LIN {X 0,Y 501.495,Z 927.191,A -85,B 0,C 180,E1 14910.89,E2 14910.89} C_VEL
LIN {X 0,Y 476.741,Z 888.568,A -85,B 0,C 180,E1 14918.992,E2 14918.992} C_VEL
LIN {X 0,Y 459.302,Z 865.995,A -85,B 0,C 180,E1 14927.264,E2 14927.264} C_VEL
LIN {X 0,Y 453.825,Z 859.085,A -85,B 0,C 180,E1 14931.559,E2 14931.559} C_VEL
LIN {X 0,Y 449.713,Z 853.483,A -85,B 0,C 180,E1 14939.969,E2 14939.969} C_VEL
LIN {X 0,Y 456.227,Z 862.461,A -85,B 0,C 180,E1 14950.385,E2 14950.385} C_VEL
LIN {X 0,Y 467.484,Z 876.849,A -85,B 0,C 180,E1 14956.99,E2 14956.99} C_VEL
LIN {X 0,Y 488.733,Z 906.336,A -85,B 0,C 180,E1 14964.926,E2 14964.926} C_VEL
LIN {X 0,Y 513.325,Z 949.109,A -85,B 0,C 180,E1 14972.183,E2 14972.183} C_VEL
LIN {X 0,Y 525.687,Z 980.917,A -85,B 0,C 180,E1 14976.061,E2 14976.061} C_VEL
LIN {X 0,Y 510.224,Z 1051.4,A -85,B 0,C 180,E1 14979.425,E2 14979.425} C_VEL
LIN {X 0,Y 490.436,Z 1119.326,A -85,B 0,C 180,E1 14984.666,E2 14984.666} C_VEL
LIN {X 0,Y 470.634,Z 1178.94,A -85,B 0,C 180,E1 14991.825,E2 14991.825} C_VEL
LIN {X 0,Y 455.077,Z 1227.051,A -85,B 0,C 180,E1 15000.689,E2 15000.689} C_VEL
LIN {X 0,Y 446.421,Z 1260.098,A -85,B 0,C 180,E1 15010.141,E2 15010.141} C_VEL
LIN {X 0,Y 443.545,Z 1278.907,A -85,B 0,C 180,E1 15019.161,E2 15019.161} C_VEL
LIN {X 0,Y 443.233,Z 1286.226,A -85,B 0,C 180,E1 15027.058,E2 15027.058} C_VEL
LIN {X 0,Y 443.148,Z 1285.182,A -85,B 0,C 180,E1 15034.908,E2 15034.908} C_VEL
LIN {X 0,Y 443.658,Z 1277.124,A -85,B 0,C 180,E1 15041.963,E2 15041.963} C_VEL
LIN {X 0,Y 437.23,Z 1269.245,A -85,B 0,C 180,E1 15046.394,E2 15046.394} C_VEL
LIN {X 0,Y 443.661,Z 1240.734,A -85,B 0,C 180,E1 15056.383,E2 15056.383} C_VEL
LIN {X 0,Y 457.28,Z 1198.235,A -85,B 0,C 180,E1 15065.684,E2 15065.684} C_VEL
LIN {X 0,Y 476.969,Z 1142.146,A -85,B 0,C 180,E1 15073.629,E2 15073.629} C_VEL
LIN {X 0,Y 497.802,Z 1076.976,A -85,B 0,C 180,E1 15079.607,E2 15079.607} C_VEL
LIN {X 0,Y 516.277,Z 1003.643,A -85,B 0,C 180,E1 15083.798,E2 15083.798} C_VEL
LIN {X 0,Y 519.992,Z 980.36,A -85,B 0,C 180,E1 15084.85,E2 15084.85} C_VEL
LIN {X 0,Y 499.484,Z 935.129,A -85,B 0,C 180,E1 15091.226,E2 15091.226} C_VEL
LIN {X 0,Y 476.703,Z 899.572,A -85,B 0,C 180,E1 15098.748,E2 15098.748} C_VEL
LIN {X 0,Y 458.796,Z 874.684,A -85,B 0,C 180,E1 15107.256,E2 15107.256} C_VEL
LIN {X 0,Y 451.996,Z 866.689,A -85,B 0,C 180,E1 15112.801,E2 15112.801} C_VEL
LIN {X 0,Y 448.923,Z 862.376,A -85,B 0,C 180,E1 15120.515,E2 15120.515} C_VEL
LIN {X 0,Y 454.937,Z 870.236,A -85,B 0,C 180,E1 15130.114,E2 15130.114} C_VEL
LIN {X 0,Y 466.224,Z 885.028,A -85,B 0,C 180,E1 15136.938,E2 15136.938} C_VEL
LIN {X 0,Y 487.537,Z 915.75,A -85,B 0,C 180,E1 15145.24,E2 15145.24} C_VEL
LIN {X 0,Y 511.002,Z 960.348,A -85,B 0,C 180,E1 15152.735,E2 15152.735} C_VEL
LIN {X 0,Y 519.263,Z 983.911,A -85,B 0,C 180,E1 15155.652,E2 15155.652} C_VEL
LIN {X 0,Y 501.618,Z 1058.051,A -85,B 0,C 180,E1 15159.562,E2 15159.562} C_VEL
LIN {X 0,Y 480.854,Z 1124.559,A -85,B 0,C 180,E1 15165.264,E2 15165.264} C_VEL
LIN {X 0,Y 460.838,Z 1181.172,A -85,B 0,C 180,E1 15172.79,E2 15172.79} C_VEL
LIN {X 0,Y 445.644,Z 1226.459,A -85,B 0,C 180,E1 15182.124,E2 15182.124} C_VEL
LIN {X 0,Y 437.765,Z 1257.62,A -85,B 0,C 180,E1 15192.467,E2 15192.467} C_VEL
LIN {X 0,Y 435.276,Z 1273.211,A -85,B 0,C 180,E1 15201.989,E2 15201.989} C_VEL
LIN {X 0,Y 435.375,Z 1277.067,A -85,B 0,C 180,E1 15210.998,E2 15210.998} C_VEL
LIN {X 0,Y 435.467,Z 1270.726,A -85,B 0,C 180,E1 15220.028,E2 15220.028} C_VEL
LIN {X 0,Y 438.618,Z 1252.212,A -85,B 0,C 180,E1 15229.701,E2 15229.701} C_VEL
LIN {X 0,Y 448.511,Z 1217.589,A -85,B 0,C 180,E1 15239.961,E2 15239.961} C_VEL
LIN {X 0,Y 464.976,Z 1169.906,A -85,B 0,C 180,E1 15248.872,E2 15248.872} C_VEL
LIN {X 0,Y 485.246,Z 1111.113,A -85,B 0,C 180,E1 15256.017,E2 15256.017} C_VEL
LIN {X 0,Y 505.549,Z 1043.955,A -85,B 0,C 180,E1 15261.223,E2 15261.223} C_VEL
LIN {X 0,Y 518.976,Z 979.558,A -85,B 0,C 180,E1 15264.58,E2 15264.58} C_VEL
LIN {X 0,Y 496.602,Z 930.952,A -85,B 0,C 180,E1 15271.706,E2 15271.706} C_VEL
LIN {X 0,Y 473.84,Z 895.17,A -85,B 0,C 180,E1 15279.593,E2 15279.593} C_VEL
LIN {X 0,Y 457.868,Z 873.617,A -85,B 0,C 180,E1 15287.532,E2 15287.532} C_VEL
LIN {X 0,Y 452.354,Z 866.791,A -85,B 0,C 180,E1 15292.017,E2 15292.017} C_VEL
LIN {X 0,Y 448.735,Z 861.449,A -85,B 0,C 180,E1 15299.969,E2 15299.969} C_VEL
LIN {X 0,Y 455.016,Z 870.359,A -85,B 0,C 180,E1 15310.231,E2 15310.231} C_VEL
LIN {X 0,Y 466.161,Z 884.963,A -85,B 0,C 180,E1 15316.877,E2 15316.877} C_VEL
LIN {X 0,Y 487.839,Z 915.843,A -85,B 0,C 180,E1 15325.159,E2 15325.159} C_VEL
LIN {X 0,Y 511.528,Z 960.138,A -85,B 0,C 180,E1 15332.514,E2 15332.514} C_VEL
LIN {X 0,Y 520.206,Z 984.714,A -85,B 0,C 180,E1 15335.473,E2 15335.473} C_VEL
LIN {X 0,Y 503.561,Z 1056.776,A -85,B 0,C 180,E1 15339.044,E2 15339.044} C_VEL
LIN {X 0,Y 483.304,Z 1123.218,A -85,B 0,C 180,E1 15344.36,E2 15344.36} C_VEL
LIN {X 0,Y 462.993,Z 1181.823,A -85,B 0,C 180,E1 15351.633,E2 15351.633} C_VEL
LIN {X 0,Y 447.269,Z 1228.623,A -85,B 0,C 180,E1 15360.551,E2 15360.551} C_VEL
LIN {X 0,Y 438.37,Z 1261.359,A -85,B 0,C 180,E1 15370.287,E2 15370.287} C_VEL
LIN {X 0,Y 435.523,Z 1280.164,A -85,B 0,C 180,E1 15379.973,E2 15379.973} C_VEL
LIN {X 0,Y 434.878,Z 1286.595,A -85,B 0,C 180,E1 15389.001,E2 15389.001} C_VEL
LIN {X 0,Y 435.311,Z 1282.6,A -85,B 0,C 180,E1 15398.01,E2 15398.01} C_VEL
LIN {X 0,Y 437.23,Z 1269.245,A -85,B 0,C 180,E1 15406.394,E2 15406.394} C_VEL
LIN {X 0,Y 431.04,Z 1259.359,A -85,B 0,C 180,E1 15410.823,E2 15410.823} C_VEL
LIN {X 0,Y 441.547,Z 1223.978,A -85,B 0,C 180,E1 15421.056,E2 15421.056} C_VEL
LIN {X 0,Y 458.603,Z 1176.1,A -85,B 0,C 180,E1 15429.877,E2 15429.877} C_VEL
LIN {X 0,Y 479.802,Z 1116.617,A -85,B 0,C 180,E1 15437.002,E2 15437.002} C_VEL
LIN {X 0,Y 500.574,Z 1049.302,A -85,B 0,C 180,E1 15442.146,E2 15442.146} C_VEL
LIN {X 0,Y 514.628,Z 984.001,A -85,B 0,C 180,E1 15445.46,E2 15445.46} C_VEL
LIN {X 0,Y 494.654,Z 938.886,A -85,B 0,C 180,E1 15452.034,E2 15452.034} C_VEL
LIN {X 0,Y 472.061,Z 902.933,A -85,B 0,C 180,E1 15460.067,E2 15460.067} C_VEL
LIN {X 0,Y 456.456,Z 881.69,A -85,B 0,C 180,E1 15468.088,E2 15468.088} C_VEL
LIN {X 0,Y 450.6,Z 874.34,A -85,B 0,C 180,E1 15473.264,E2 15473.264} C_VEL
LIN {X 0,Y 447.949,Z 870.312,A -85,B 0,C 180,E1 15480.517,E2 15480.517} C_VEL
LIN {X 0,Y 453.804,Z 878.246,A -85,B 0,C 180,E1 15490.018,E2 15490.018} C_VEL
LIN {X 0,Y 464.959,Z 893.354,A -85,B 0,C 180,E1 15496.925,E2 15496.925} C_VEL
LIN {X 0,Y 485.315,Z 923.772,A -85,B 0,C 180,E1 15505.11,E2 15505.11} C_VEL
LIN {X 0,Y 506.806,Z 966.395,A -85,B 0,C 180,E1 15512.381,E2 15512.381} C_VEL
LIN {X 0,Y 513.595,Z 988.518,A -85,B 0,C 180,E1 15515.105,E2 15515.105} C_VEL
LIN {X 0,Y 495.036,Z 1062.693,A -85,B 0,C 180,E1 15519.15,E2 15519.15} C_VEL
LIN {X 0,Y 473.79,Z 1127.945,A -85,B 0,C 180,E1 15524.925,E2 15524.925} C_VEL
LIN {X 0,Y 453.117,Z 1184.181,A -85,B 0,C 180,E1 15532.654,E2 15532.654} C_VEL
LIN {X 0,Y 437.576,Z 1228.757,A -85,B 0,C 180,E1 15542.205,E2 15542.205} C_VEL
LIN {X 0,Y 429.704,Z 1258.601,A -85,B 0,C 180,E1 15552.543,E2 15552.543} C_VEL
LIN {X 0,Y 427.308,Z 1273.298,A -85,B 0,C 180,E1 15561.839,E2 15561.839} C_VEL
LIN {X 0,Y 427.391,Z 1277.155,A -85,B 0,C 180,E1 15571.017,E2 15571.017} C_VEL
LIN {X 0,Y 427.483,Z 1270.816,A -85,B 0,C 180,E1 15580.217,E2 15580.217} C_VEL
LIN {X 0,Y 431.216,Z 1251.295,A -85,B 0,C 180,E1 15590.462,E2 15590.462} C_VEL
LIN {X 0,Y 441.691,Z 1216.518,A -85,B 0,C 180,E1 15600.781,E2 15600.781} C_VEL
LIN {X 0,Y 458.714,Z 1169.437,A -85,B 0,C 180,E1 15609.614,E2 15609.614} C_VEL
LIN {X 0,Y 479.414,Z 1111.581,A -85,B 0,C 180,E1 15616.691,E2 15616.691} C_VEL
LIN {X 0,Y 500.553,Z 1043.74,A -85,B 0,C 180,E1 15621.972,E2 15621.972} C_VEL
LIN {X 0,Y 513.747,Z 983.715,A -85,B 0,C 180,E1 15625.133,E2 15625.133} C_VEL
LIN {X 0,Y 492.652,Z 936.614,A -85,B 0,C 180,E1 15632.236,E2 15632.236} C_VEL
LIN {X 0,Y 471.152,Z 901.763,A -85,B 0,C 180,E1 15640.147,E2 15640.147} C_VEL
LIN {X 0,Y 456.144,Z 880.962,A -85,B 0,C 180,E1 15647.999,E2 15647.999} C_VEL
LIN {X 0,Y 450.912,Z 874.489,A -85,B 0,C 180,E1 15652.478,E2 15652.478} C_VEL
LIN {X 0,Y 447.759,Z 869.4,A -85,B 0,C 180,E1 15659.969,E2 15659.969} C_VEL
LIN {X 0,Y 453.811,Z 878.238,A -85,B 0,C 180,E1 15670.076,E2 15670.076} C_VEL
LIN {X 0,Y 465.304,Z 893.818,A -85,B 0,C 180,E1 15677.032,E2 15677.032} C_VEL
LIN {X 0,Y 485.785,Z 924.152,A -85,B 0,C 180,E1 15685.088,E2 15685.088} C_VEL
LIN {X 0,Y 508.014,Z 967.632,A -85,B 0,C 180,E1 15692.348,E2 15692.348} C_VEL
LIN {X 0,Y 515.001,Z 987.452,A -85,B 0,C 180,E1 15694.839,E2 15694.839} C_VEL
LIN {X 0,Y 498.134,Z 1057.756,A -85,B 0,C 180,E1 15698.378,E2 15698.378} C_VEL
LIN {X 0,Y 477.644,Z 1122.698,A -85,B 0,C 180,E1 15703.601,E2 15703.601} C_VEL
LIN {X 0,Y 456.424,Z 1181.853,A -85,B 0,C 180,E1 15711.001,E2 15711.001} C_VEL
LIN {X 0,Y 439.967,Z 1228.53,A -85,B 0,C 180,E1 15720.013,E2 15720.013} C_VEL
LIN {X 0,Y 430.816,Z 1260.254,A -85,B 0,C 180,E1 15729.524,E2 15729.524} C_VEL
LIN {X 0,Y 427.57,Z 1278.729,A -85,B 0,C 180,E1 15738.751,E2 15738.751} C_VEL
LIN {X 0,Y 427.242,Z 1286.051,A -85,B 0,C 180,E1 15746.948,E2 15746.948} C_VEL
LIN {X 0,Y 427.152,Z 1285.007,A -85,B 0,C 180,E1 15755.092,E2 15755.092} C_VEL
LIN {X 0,Y 428.304,Z 1273.725,A -85,B 0,C 180,E1 15764.351,E2 15764.351} C_VEL
LIN {X 0,Y 431.04,Z 1259.359,A -85,B 0,C 180,E1 15770.823,E2 15770.823} C_VEL
LIN {X 0,Y 426.882,Z 1247.494,A -85,B 0,C 180,E1 15775.272,E2 15775.272} C_VEL
LIN {X 0,Y 440.642,Z 1206.475,A -85,B 0,C 180,E1 15785.339,E2 15785.339} C_VEL
LIN {X 0,Y 460.695,Z 1153.533,A -85,B 0,C 180,E1 15793.646,E2 15793.646} C_VEL
LIN {X 0,Y 483.118,Z 1089.437,A -85,B 0,C 180,E1 15800.131,E2 15800.131} C_VEL
LIN {X 0,Y 503.794,Z 1017.149,A -85,B 0,C 180,E1 15804.635,E2 15804.635} C_VEL
LIN {X 0,Y 509.483,Z 987.866,A -85,B 0,C 180,E1 15806.041,E2 15806.041} C_VEL
LIN {X 0,Y 490.493,Z 944.188,A -85,B 0,C 180,E1 15812.634,E2 15812.634} C_VEL
LIN {X 0,Y 469.524,Z 909.664,A -85,B 0,C 180,E1 15820.569,E2 15820.569} C_VEL
LIN {X 0,Y 454.853,Z 889.166,A -85,B 0,C 180,E1 15828.488,E2 15828.488} C_VEL
LIN {X 0,Y 449.46,Z 882.146,A -85,B 0,C 180,E1 15833.454,E2 15833.454} C_VEL
LIN {X 0,Y 447.012,Z 878.319,A -85,B 0,C 180,E1 15841.004,E2 15841.004} C_VEL
LIN {X 0,Y 452.674,Z 886.24,A -85,B 0,C 180,E1 15849.921,E2 15849.921} C_VEL
LIN {X 0,Y 463.901,Z 901.925,A -85,B 0,C 180,E1 15857.026,E2 15857.026} C_VEL
LIN {X 0,Y 483.881,Z 933.368,A -85,B 0,C 180,E1 15865.366,E2 15865.366} C_VEL
LIN {X 0,Y 503.989,Z 976.276,A -85,B 0,C 180,E1 15872.584,E2 15872.584} C_VEL
LIN {X 0,Y 508.188,Z 992.307,A -85,B 0,C 180,E1 15874.517,E2 15874.517} C_VEL
LIN {X 0,Y 488.734,Z 1066.589,A -85,B 0,C 180,E1 15878.677,E2 15878.677} C_VEL
LIN {X 0,Y 466.613,Z 1131.769,A -85,B 0,C 180,E1 15884.628,E2 15884.628} C_VEL
LIN {X 0,Y 445.395,Z 1187.175,A -85,B 0,C 180,E1 15892.51,E2 15892.51} C_VEL
LIN {X 0,Y 429.653,Z 1230.659,A -85,B 0,C 180,E1 15902.183,E2 15902.183} C_VEL
LIN {X 0,Y 421.726,Z 1259.366,A -85,B 0,C 180,E1 15912.523,E2 15912.523} C_VEL
LIN {X 0,Y 419.26,Z 1274.237,A -85,B 0,C 180,E1 15922.727,E2 15922.727} C_VEL
LIN {X 0,Y 419.385,Z 1277.242,A -85,B 0,C 180,E1 15931.036,E2 15931.036} C_VEL
LIN {X 0,Y 419.52,Z 1270.906,A -85,B 0,C 180,E1 15940.413,E2 15940.413} C_VEL
LIN {X 0,Y 423.479,Z 1251.584,A -85,B 0,C 180,E1 15950.771,E2 15950.771} C_VEL
LIN {X 0,Y 434.477,Z 1216.776,A -85,B 0,C 180,E1 15961.305,E2 15961.305} C_VEL
LIN {X 0,Y 452.135,Z 1169.99,A -85,B 0,C 180,E1 15970.217,E2 15970.217} C_VEL
LIN {X 0,Y 473.478,Z 1112.488,A -85,B 0,C 180,E1 15977.338,E2 15977.338} C_VEL
LIN {X 0,Y 495.08,Z 1045.523,A -85,B 0,C 180,E1 15982.61,E2 15982.61} C_VEL
LIN {X 0,Y 508.615,Z 988.345,A -85,B 0,C 180,E1 15985.617,E2 15985.617} C_VEL
LIN {X 0,Y 488.905,Z 942.436,A -85,B 0,C 180,E1 15992.727,E2 15992.727} C_VEL
LIN {X 0,Y 468.545,Z 908.479,A -85,B 0,C 180,E1 16000.647,E2 16000.647} C_VEL
LIN {X 0,Y 454.199,Z 887.857,A -85,B 0,C 180,E1 16008.652,E2 16008.652} C_VEL
LIN {X 0,Y 449.303,Z 881.947,A -85,B 0,C 180,E1 16013.182,E2 16013.182} C_VEL
LIN {X 0,Y 446.773,Z 877.479,A -85,B 0,C 180,E1 16020.212,E2 16020.212} C_VEL
LIN {X 0,Y 452.748,Z 886.334,A -85,B 0,C 180,E1 16030.039,E2 16030.039} C_VEL
LIN {X 0,Y 466.383,Z 904.689,A -85,B 0,C 180,E1 16038.09,E2 16038.09} C_VEL
LIN {X 0,Y 488.354,Z 940.813,A -85,B 0,C 180,E1 16046.7,E2 16046.7} C_VEL
LIN {X 0,Y 508.381,Z 985.693,A -85,B 0,C 180,E1 16053.642,E2 16053.642} C_VEL
LIN {X 0,Y 508.76,Z 994.841,A -85,B 0,C 180,E1 16054.379,E2 16054.379} C_VEL
LIN {X 0,Y 490.55,Z 1066.473,A -85,B 0,C 180,E1 16058.216,E2 16058.216} C_VEL
LIN {X 0,Y 468.734,Z 1131.664,A -85,B 0,C 180,E1 16063.802,E2 16063.802} C_VEL
LIN {X 0,Y 447.224,Z 1188.791,A -85,B 0,C 180,E1 16071.457,E2 16071.457} C_VEL
LIN {X 0,Y 431.31,Z 1232.689,A -85,B 0,C 180,E1 16080.511,E2 16080.511} C_VEL
LIN {X 0,Y 422.21,Z 1263.877,A -85,B 0,C 180,E1 16090.594,E2 16090.594} C_VEL
LIN {X 0,Y 419.508,Z 1281.211,A -85,B 0,C 180,E1 16100.638,E2 16100.638} C_VEL
LIN {X 0,Y 418.904,Z 1286.42,A -85,B 0,C 180,E1 16108.963,E2 16108.963} C_VEL
LIN {X 0,Y 419.371,Z 1282.424,A -85,B 0,C 180,E1 16118.317,E2 16118.317} C_VEL
LIN {X 0,Y 422.02,Z 1265.061,A -85,B 0,C 180,E1 16128.87,E2 16128.87} C_VEL
LIN {X 0,Y 426.882,Z 1247.494,A -85,B 0,C 180,E1 16135.272,E2 16135.272} C_VEL
LIN {X 0,Y 423.428,Z 1233.999,A -85,B 0,C 180,E1 16139.672,E2 16139.672} C_VEL
LIN {X 0,Y 440.551,Z 1189.039,A -85,B 0,C 180,E1 16149.169,E2 16149.169} C_VEL
LIN {X 0,Y 462.996,Z 1131.691,A -85,B 0,C 180,E1 16156.933,E2 16156.933} C_VEL
LIN {X 0,Y 485.073,Z 1067.793,A -85,B 0,C 180,E1 16162.458,E2 16162.458} C_VEL
LIN {X 0,Y 504.343,Z 993.938,A -85,B 0,C 180,E1 16166.442,E2 16166.442} C_VEL
LIN {X 0,Y 488.8,Z 954.294,A -85,B 0,C 180,E1 16172.349,E2 16172.349} C_VEL
LIN {X 0,Y 468.027,Z 917.942,A -85,B 0,C 180,E1 16180.504,E2 16180.504} C_VEL
LIN {X 0,Y 453.214,Z 896.694,A -85,B 0,C 180,E1 16188.813,E2 16188.813} C_VEL
LIN {X 0,Y 448.058,Z 889.725,A -85,B 0,C 180,E1 16193.958,E2 16193.958} C_VEL
LIN {X 0,Y 446.055,Z 886.405,A -85,B 0,C 180,E1 16201.25,E2 16201.25} C_VEL
LIN {X 0,Y 451.459,Z 894.286,A -85,B 0,C 180,E1 16209.887,E2 16209.887} C_VEL
LIN {X 0,Y 464.308,Z 912.347,A -85,B 0,C 180,E1 16217.93,E2 16217.93} C_VEL
LIN {X 0,Y 484.467,Z 947.242,A -85,B 0,C 180,E1 16226.442,E2 16226.442} C_VEL
LIN {X 0,Y 502.784,Z 991.315,A -85,B 0,C 180,E1 16233.524,E2 16233.524} C_VEL
LIN {X 0,Y 484.988,Z 1062.482,A -85,B 0,C 180,E1 16237.623,E2 16237.623} C_VEL
LIN {X 0,Y 462.083,Z 1128.444,A -85,B 0,C 180,E1 16243.503,E2 16243.503} C_VEL
LIN {X 0,Y 439.649,Z 1184.938,A -85,B 0,C 180,E1 16251.429,E2 16251.429} C_VEL
LIN {X 0,Y 422.94,Z 1228.585,A -85,B 0,C 180,E1 16261.049,E2 16261.049} C_VEL
LIN {X 0,Y 414.085,Z 1258.777,A -85,B 0,C 180,E1 16271.862,E2 16271.862} C_VEL
LIN {X 0,Y 411.264,Z 1274.325,A -85,B 0,C 180,E1 16282.585,E2 16282.585} C_VEL
LIN {X 0,Y 411.383,Z 1277.33,A -85,B 0,C 180,E1 16291.056,E2 16291.056} C_VEL
LIN {X 0,Y 411.551,Z 1270.995,A -85,B 0,C 180,E1 16300.617,E2 16300.617} C_VEL
LIN {X 0,Y 416.072,Z 1250.837,A -85,B 0,C 180,E1 16311.512,E2 16311.512} C_VEL
LIN {X 0,Y 427.519,Z 1216.355,A -85,B 0,C 180,E1 16322.016,E2 16322.016} C_VEL
LIN {X 0,Y 446.398,Z 1168.492,A -85,B 0,C 180,E1 16331.164,E2 16331.164} C_VEL
LIN {X 0,Y 468.812,Z 1110.065,A -85,B 0,C 180,E1 16338.341,E2 16338.341} C_VEL
LIN {X 0,Y 491.28,Z 1041.862,A -85,B 0,C 180,E1 16343.603,E2 16343.603} C_VEL
LIN {X 0,Y 503.126,Z 991.836,A -85,B 0,C 180,E1 16346.269,E2 16346.269} C_VEL
LIN {X 0,Y 484.214,Z 946.383,A -85,B 0,C 180,E1 16353.563,E2 16353.563} C_VEL
LIN {X 0,Y 463.692,Z 911.268,A -85,B 0,C 180,E1 16362.23,E2 16362.23} C_VEL
LIN {X 0,Y 450.421,Z 891.105,A -85,B 0,C 180,E1 16371.007,E2 16371.007} C_VEL
LIN {X 0,Y 445.805,Z 885.314,A -85,B 0,C 180,E1 16379.968,E2 16379.968} C_VEL
LIN {X 0,Y 451.434,Z 894.164,A -85,B 0,C 180,E1 16389.885,E2 16389.885} C_VEL
LIN {X 0,Y 464.661,Z 912.823,A -85,B 0,C 180,E1 16397.975,E2 16397.975} C_VEL
LIN {X 0,Y 485.086,Z 947.542,A -85,B 0,C 180,E1 16406.358,E2 16406.358} C_VEL
LIN {X 0,Y 503.892,Z 991.626,A -85,B 0,C 180,E1 16413.313,E2 16413.313} C_VEL
LIN {X 0,Y 485.622,Z 1065.969,A -85,B 0,C 180,E1 16417.422,E2 16417.422} C_VEL
LIN {X 0,Y 463.028,Z 1131.567,A -85,B 0,C 180,E1 16423.06,E2 16423.06} C_VEL
LIN {X 0,Y 440.549,Z 1189.028,A -85,B 0,C 180,E1 16430.834,E2 16430.834} C_VEL
LIN {X 0,Y 423.318,Z 1234.563,A -85,B 0,C 180,E1 16440.489,E2 16440.489} C_VEL
LIN {X 0,Y 414.165,Z 1264.967,A -85,B 0,C 180,E1 16450.758,E2 16450.758} C_VEL
LIN {X 0,Y 411.511,Z 1281.122,A -85,B 0,C 180,E1 16460.454,E2 16460.454} C_VEL
LIN {X 0,Y 410.91,Z 1286.332,A -85,B 0,C 180,E1 16468.943,E2 16468.943} C_VEL
LIN {X 0,Y 411.413,Z 1282.336,A -85,B 0,C 180,E1 16478.479,E2 16478.479} C_VEL
LIN {X 0,Y 413.973,Z 1266.131,A -85,B 0,C 180,E1 16488.696,E2 16488.696} C_VEL
LIN {X 0,Y 422.523,Z 1236.53,A -85,B 0,C 180,E1 16498.983,E2 16498.983} C_VEL
LIN {X 0,Y 423.428,Z 1233.999,A -85,B 0,C 180,E1 16499.672,E2 16499.672} C_VEL
LIN {X 0,Y 422.311,Z 1218.571,A -85,B 0,C 180,E1 16504.014,E2 16504.014} C_VEL
LIN {X 0,Y 442.304,Z 1169.254,A -85,B 0,C 180,E1 16512.956,E2 16512.956} C_VEL
LIN {X 0,Y 465.691,Z 1109.301,A -85,B 0,C 180,E1 16519.932,E2 16519.932} C_VEL
LIN {X 0,Y 488.342,Z 1040.282,A -85,B 0,C 180,E1 16524.957,E2 16524.957} C_VEL
LIN {X 0,Y 498.704,Z 994.718,A -85,B 0,C 180,E1 16527.358,E2 16527.358} C_VEL
LIN {X 0,Y 481.274,Z 952.634,A -85,B 0,C 180,E1 16534.229,E2 16534.229} C_VEL
LIN {X 0,Y 461.467,Z 918.61,A -85,B 0,C 180,E1 16542.884,E2 16542.884} C_VEL
LIN {X 0,Y 448.865,Z 898.934,A -85,B 0,C 180,E1 16551.773,E2 16551.773} C_VEL
LIN {X 0,Y 444.924,Z 894.163,A -85,B 0,C 180,E1 16561.009,E2 16561.009} C_VEL
LIN {X 0,Y 450.158,Z 902.219,A -85,B 0,C 180,E1 16569.794,E2 16569.794} C_VEL
LIN {X 0,Y 462.509,Z 920.585,A -85,B 0,C 180,E1 16577.879,E2 16577.879} C_VEL
LIN {X 0,Y 481.234,Z 954.461,A -85,B 0,C 180,E1 16586.221,E2 16586.221} C_VEL
LIN {X 0,Y 498.024,Z 996.772,A -85,B 0,C 180,E1 16593.133,E2 16593.133} C_VEL
LIN {X 0,Y 477.643,Z 1069.957,A -85,B 0,C 180,E1 16597.376,E2 16597.376} C_VEL
LIN {X 0,Y 454.316,Z 1133.915,A -85,B 0,C 180,E1 16603.363,E2 16603.363} C_VEL
LIN {X 0,Y 431.886,Z 1188.084,A -85,B 0,C 180,E1 16611.285,E2 16611.285} C_VEL
LIN {X 0,Y 414.801,Z 1231.268,A -85,B 0,C 180,E1 16621.228,E2 16621.228} C_VEL
LIN {X 0,Y 405.965,Z 1260.2,A -85,B 0,C 180,E1 16632.146,E2 16632.146} C_VEL
LIN {X 0,Y 403.278,Z 1274.412,A -85,B 0,C 180,E1 16642.437,E2 16642.437} C_VEL
LIN {X 0,Y 403.376,Z 1277.418,A -85,B 0,C 180,E1 16651.077,E2 16651.077} C_VEL
LIN {X 0,Y 403.618,Z 1271.084,A -85,B 0,C 180,E1 16660.828,E2 16660.828} C_VEL
LIN {X 0,Y 408.433,Z 1250.929,A -85,B 0,C 180,E1 16671.935,E2 16671.935} C_VEL
LIN {X 0,Y 420.579,Z 1215.98,A -85,B 0,C 180,E1 16682.743,E2 16682.743} C_VEL
LIN {X 0,Y 440.126,Z 1168.587,A -85,B 0,C 180,E1 16691.882,E2 16691.882} C_VEL
LIN {X 0,Y 463.328,Z 1110.188,A -85,B 0,C 180,E1 16699.105,E2 16699.105} C_VEL
LIN {X 0,Y 486.461,Z 1041.967,A -85,B 0,C 180,E1 16704.379,E2 16704.379} C_VEL
LIN {X 0,Y 497.738,Z 995.471,A -85,B 0,C 180,E1 16706.918,E2 16706.918} C_VEL
LIN {X 0,Y 479.912,Z 951.543,A -85,B 0,C 180,E1 16714.211,E2 16714.211} C_VEL
LIN {X 0,Y 461.361,Z 918.547,A -85,B 0,C 180,E1 16722.569,E2 16722.569} C_VEL
LIN {X 0,Y 449.003,Z 898.935,A -85,B 0,C 180,E1 16731.223,E2 16731.223} C_VEL
LIN {X 0,Y 444.71,Z 893.249,A -85,B 0,C 180,E1 16739.968,E2 16739.968} C_VEL
LIN {X 0,Y 450.126,Z 902.119,A -85,B 0,C 180,E1 16749.792,E2 16749.792} C_VEL
LIN {X 0,Y 462.861,Z 921.046,A -85,B 0,C 180,E1 16757.924,E2 16757.924} C_VEL
LIN {X 0,Y 482.023,Z 954.851,A -85,B 0,C 180,E1 16766.159,E2 16766.159} C_VEL
LIN {X 0,Y 499.016,Z 996.731,A -85,B 0,C 180,E1 16772.88,E2 16772.88} C_VEL
LIN {X 0,Y 479.138,Z 1070.596,A -85,B 0,C 180,E1 16776.977,E2 16776.977} C_VEL
LIN {X 0,Y 456.165,Z 1134.474,A -85,B 0,C 180,E1 16782.631,E2 16782.631} C_VEL
LIN {X 0,Y 433.009,Z 1191.422,A -85,B 0,C 180,E1 16790.569,E2 16790.569} C_VEL
LIN {X 0,Y 415.292,Z 1236.436,A -85,B 0,C 180,E1 16800.463,E2 16800.463} C_VEL
LIN {X 0,Y 406.085,Z 1266.036,A -85,B 0,C 180,E1 16810.927,E2 16810.927} C_VEL
LIN {X 0,Y 403.479,Z 1282.246,A -85,B 0,C 180,E1 16821.353,E2 16821.353} C_VEL
LIN {X 0,Y 402.911,Z 1286.245,A -85,B 0,C 180,E1 16828.922,E2 16828.922} C_VEL
LIN {X 0,Y 403.45,Z 1282.248,A -85,B 0,C 180,E1 16838.647,E2 16838.647} C_VEL
LIN {X 0,Y 406.135,Z 1266.041,A -85,B 0,C 180,E1 16849.07,E2 16849.07} C_VEL
LIN {X 0,Y 415.218,Z 1236.44,A -85,B 0,C 180,E1 16859.543,E2 16859.543} C_VEL
LIN {X 0,Y 422.311,Z 1218.571,A -85,B 0,C 180,E1 16864.014,E2 16864.014} C_VEL
LIN {X 0,Y 422.196,Z 1201.624,A -85,B 0,C 180,E1 16868.249,E2 16868.249} C_VEL
LIN {X 0,Y 445.536,Z 1146.969,A -85,B 0,C 180,E1 16876.683,E2 16876.683} C_VEL
LIN {X 0,Y 469.504,Z 1084.292,A -85,B 0,C 180,E1 16882.829,E2 16882.829} C_VEL
LIN {X 0,Y 491.258,Z 1012,A -85,B 0,C 180,E1 16887.214,E2 16887.214} C_VEL
LIN {X 0,Y 493.425,Z 998.431,A -85,B 0,C 180,E1 16888.004,E2 16888.004} C_VEL
LIN {X 0,Y 476.815,Z 957.45,A -85,B 0,C 180,E1 16894.959,E2 16894.959} C_VEL
LIN {X 0,Y 458.713,Z 925.318,A -85,B 0,C 180,E1 16903.459,E2 16903.459} C_VEL
LIN {X 0,Y 447.215,Z 906.67,A -85,B 0,C 180,E1 16912.233,E2 16912.233} C_VEL
LIN {X 0,Y 443.765,Z 902.11,A -85,B 0,C 180,E1 16921.011,E2 16921.011} C_VEL
LIN {X 0,Y 448.781,Z 910.213,A -85,B 0,C 180,E1 16929.763,E2 16929.763} C_VEL
LIN {X 0,Y 460.839,Z 929.219,A -85,B 0,C 180,E1 16937.965,E2 16937.965} C_VEL
LIN {X 0,Y 478.03,Z 961.714,A -85,B 0,C 180,E1 16946.005,E2 16946.005} C_VEL
LIN {X 0,Y 492.827,Z 1001.476,A -85,B 0,C 180,E1 16952.587,E2 16952.587} C_VEL
LIN {X 0,Y 471.03,Z 1074.986,A -85,B 0,C 180,E1 16956.946,E2 16956.946} C_VEL
LIN {X 0,Y 446.821,Z 1138.601,A -85,B 0,C 180,E1 16963.137,E2 16963.137} C_VEL
LIN {X 0,Y 423.331,Z 1193.094,A -85,B 0,C 180,E1 16971.513,E2 16971.513} C_VEL
LIN {X 0,Y 406.223,Z 1234.824,A -85,B 0,C 180,E1 16981.729,E2 16981.729} C_VEL
LIN {X 0,Y 397.907,Z 1261.186,A -85,B 0,C 180,E1 16992.224,E2 16992.224} C_VEL
LIN {X 0,Y 395.288,Z 1274.5,A -85,B 0,C 180,E1 17002.283,E2 17002.283} C_VEL
LIN {X 0,Y 395.383,Z 1277.505,A -85,B 0,C 180,E1 17011.099,E2 17011.099} C_VEL
LIN {X 0,Y 395.678,Z 1271.19,A -85,B 0,C 180,E1 17021.033,E2 17021.033} C_VEL
LIN {X 0,Y 400.778,Z 1250.918,A -85,B 0,C 180,E1 17032.422,E2 17032.422} C_VEL
LIN {X 0,Y 413.514,Z 1216.074,A -85,B 0,C 180,E1 17043.375,E2 17043.375} C_VEL
LIN {X 0,Y 433.91,Z 1168.768,A -85,B 0,C 180,E1 17052.604,E2 17052.604} C_VEL
LIN {X 0,Y 457.879,Z 1110.501,A -85,B 0,C 180,E1 17059.864,E2 17059.864} C_VEL
LIN {X 0,Y 481.386,Z 1043.243,A -85,B 0,C 180,E1 17065.094,E2 17065.094} C_VEL
LIN {X 0,Y 492.38,Z 998.95,A -85,B 0,C 180,E1 17067.6,E2 17067.6} C_VEL
LIN {X 0,Y 475.366,Z 955.901,A -85,B 0,C 180,E1 17075.017,E2 17075.017} C_VEL
LIN {X 0,Y 458.414,Z 924.969,A -85,B 0,C 180,E1 17083.246,E2 17083.246} C_VEL
LIN {X 0,Y 447.595,Z 906.733,A -85,B 0,C 180,E1 17091.441,E2 17091.441} C_VEL
LIN {X 0,Y 443.551,Z 901.348,A -85,B 0,C 180,E1 17100.458,E2 17100.458} C_VEL
LIN {X 0,Y 448.89,Z 910.227,A -85,B 0,C 180,E1 17109.819,E2 17109.819} C_VEL
LIN {X 0,Y 461.536,Z 930.004,A -85,B 0,C 180,E1 17118.121,E2 17118.121} C_VEL
LIN {X 0,Y 479.321,Z 963.285,A -85,B 0,C 180,E1 17126.161,E2 17126.161} C_VEL
LIN {X 0,Y 493.686,Z 1001.873,A -85,B 0,C 180,E1 17132.353,E2 17132.353} C_VEL
LIN {X 0,Y 473.205,Z 1073.57,A -85,B 0,C 180,E1 17136.399,E2 17136.399} C_VEL
LIN {X 0,Y 449.274,Z 1137.556,A -85,B 0,C 180,E1 17142.211,E2 17142.211} C_VEL
LIN {X 0,Y 425.837,Z 1192.969,A -85,B 0,C 180,E1 17150.143,E2 17150.143} C_VEL
LIN {X 0,Y 408.021,Z 1236.343,A -85,B 0,C 180,E1 17159.883,E2 17159.883} C_VEL
LIN {X 0,Y 398.285,Z 1265.945,A -85,B 0,C 180,E1 17170.539,E2 17170.539} C_VEL
LIN {X 0,Y 395.497,Z 1282.158,A -85,B 0,C 180,E1 17181.177,E2 17181.177} C_VEL
LIN {X 0,Y 394.926,Z 1286.157,A -85,B 0,C 180,E1 17188.9,E2 17188.9} C_VEL
LIN {X 0,Y 395.473,Z 1282.16,A -85,B 0,C 180,E1 17198.823,E2 17198.823} C_VEL
LIN {X 0,Y 398.32,Z 1265.952,A -85,B 0,C 180,E1 17209.459,E2 17209.459} C_VEL
LIN {X 0,Y 407.932,Z 1236.349,A -85,B 0,C 180,E1 17220.124,E2 17220.124} C_VEL
LIN {X 0,Y 422.196,Z 1201.624,A -85,B 0,C 180,E1 17228.249,E2 17228.249} C_VEL
LIN {X 0,Y 424.032,Z 1182.881,A -85,B 0,C 180,E1 17232.326,E2 17232.326} C_VEL
LIN {X 0,Y 449.332,Z 1123.987,A -85,B 0,C 180,E1 17240.062,E2 17240.062} C_VEL
LIN {X 0,Y 473.541,Z 1058.255,A -85,B 0,C 180,E1 17245.455,E2 17245.455} C_VEL
LIN {X 0,Y 488.206,Z 1001.997,A -85,B 0,C 180,E1 17248.676,E2 17248.676} C_VEL
LIN {X 0,Y 472.128,Z 961.302,A -85,B 0,C 180,E1 17255.867,E2 17255.867} C_VEL
LIN {X 0,Y 454.67,Z 929.554,A -85,B 0,C 180,E1 17264.851,E2 17264.851} C_VEL
LIN {X 0,Y 444.725,Z 913.866,A -85,B 0,C 180,E1 17273.421,E2 17273.421} C_VEL
LIN {X 0,Y 442.505,Z 910.022,A -85,B 0,C 180,E1 17281.014,E2 17281.014} C_VEL
LIN {X 0,Y 447.131,Z 918.074,A -85,B 0,C 180,E1 17289.676,E2 17289.676} C_VEL
LIN {X 0,Y 458.843,Z 937.471,A -85,B 0,C 180,E1 17297.997,E2 17297.997} C_VEL
LIN {X 0,Y 475.259,Z 970.215,A -85,B 0,C 180,E1 17306.067,E2 17306.067} C_VEL
LIN {X 0,Y 487.416,Z 1005.685,A -85,B 0,C 180,E1 17311.976,E2 17311.976} C_VEL
LIN {X 0,Y 465.08,Z 1077.889,A -85,B 0,C 180,E1 17316.361,E2 17316.361} C_VEL
LIN {X 0,Y 440.319,Z 1140.601,A -85,B 0,C 180,E1 17322.592,E2 17322.592} C_VEL
LIN {X 0,Y 416.472,Z 1193.877,A -85,B 0,C 180,E1 17330.936,E2 17330.936} C_VEL
LIN {X 0,Y 398.849,Z 1234.914,A -85,B 0,C 180,E1 17341.158,E2 17341.158} C_VEL
LIN {X 0,Y 389.604,Z 1262.675,A -85,B 0,C 180,E1 17352.67,E2 17352.67} C_VEL
LIN {X 0,Y 387.319,Z 1274.588,A -85,B 0,C 180,E1 17362.123,E2 17362.123} C_VEL
LIN {X 0,Y 387.291,Z 1277.483,A -85,B 0,C 180,E1 17371.854,E2 17371.854} C_VEL
LIN {X 0,Y 387.998,Z 1269.933,A -85,B 0,C 180,E1 17382.414,E2 17382.414} C_VEL
LIN {X 0,Y 393.711,Z 1248.76,A -85,B 0,C 180,E1 17393.857,E2 17393.857} C_VEL
LIN {X 0,Y 407.882,Z 1212.849,A -85,B 0,C 180,E1 17404.866,E2 17404.866} C_VEL
LIN {X 0,Y 430.021,Z 1163.814,A -85,B 0,C 180,E1 17414.148,E2 17414.148} C_VEL
LIN {X 0,Y 455.325,Z 1103.919,A -85,B 0,C 180,E1 17421.296,E2 17421.296} C_VEL
LIN {X 0,Y 479.183,Z 1035.362,A -85,B 0,C 180,E1 17426.375,E2 17426.375} C_VEL
LIN {X 0,Y 487.323,Z 1003.169,A -85,B 0,C 180,E1 17428.18,E2 17428.18} C_VEL
LIN {X 0,Y 471.02,Z 960.5,A -85,B 0,C 180,E1 17435.788,E2 17435.788} C_VEL
LIN {X 0,Y 454.775,Z 930.104,A -85,B 0,C 180,E1 17444.304,E2 17444.304} C_VEL
LIN {X 0,Y 445.384,Z 914.245,A -85,B 0,C 180,E1 17452.137,E2 17452.137} C_VEL
LIN {X 0,Y 442.332,Z 909.262,A -85,B 0,C 180,E1 17460.459,E2 17460.459} C_VEL
LIN {X 0,Y 447.176,Z 917.974,A -85,B 0,C 180,E1 17469.672,E2 17469.672} C_VEL
LIN {X 0,Y 459.345,Z 937.842,A -85,B 0,C 180,E1 17478.041,E2 17478.041} C_VEL
LIN {X 0,Y 476.088,Z 970.479,A -85,B 0,C 180,E1 17485.952,E2 17485.952} C_VEL
LIN {X 0,Y 488.249,Z 1006.475,A -85,B 0,C 180,E1 17491.741,E2 17491.741} C_VEL
LIN {X 0,Y 466.697,Z 1078.421,A -85,B 0,C 180,E1 17495.942,E2 17495.942} C_VEL
LIN {X 0,Y 441.611,Z 1142.652,A -85,B 0,C 180,E1 17502.014,E2 17502.014} C_VEL
LIN {X 0,Y 416.905,Z 1198.665,A -85,B 0,C 180,E1 17510.463,E2 17510.463} C_VEL
LIN {X 0,Y 398.84,Z 1241.203,A -85,B 0,C 180,E1 17520.725,E2 17520.725} C_VEL
LIN {X 0,Y 389.874,Z 1268.872,A -85,B 0,C 180,E1 17531.634,E2 17531.634} C_VEL
LIN {X 0,Y 387.327,Z 1282.947,A -85,B 0,C 180,E1 17542.123,E2 17542.123} C_VEL
LIN {X 0,Y 386.819,Z 1286.069,A -85,B 0,C 180,E1 17551.123,E2 17551.123} C_VEL
LIN {X 0,Y 387.667,Z 1279.633,A -85,B 0,C 180,E1 17561.28,E2 17561.28} C_VEL
LIN {X 0,Y 391.978,Z 1260.935,A -85,B 0,C 180,E1 17572.111,E2 17572.111} C_VEL
LIN {X 0,Y 404.77,Z 1226.985,A -85,B 0,C 180,E1 17583.226,E2 17583.226} C_VEL
LIN {X 0,Y 424.032,Z 1182.881,A -85,B 0,C 180,E1 17592.326,E2 17592.326} C_VEL
LIN {X 0,Y 427.2,Z 1162.447,A -85,B 0,C 180,E1 17596.219,E2 17596.219} C_VEL
LIN {X 0,Y 453.256,Z 1100.893,A -85,B 0,C 180,E1 17603.101,E2 17603.101} C_VEL
LIN {X 0,Y 477.709,Z 1030.052,A -85,B 0,C 180,E1 17607.921,E2 17607.921} C_VEL
LIN {X 0,Y 483.448,Z 1007.03,A -85,B 0,C 180,E1 17609.154,E2 17609.154} C_VEL
LIN {X 0,Y 468.239,Z 967.041,A -85,B 0,C 180,E1 17616.436,E2 17616.436} C_VEL
LIN {X 0,Y 451.523,Z 935.188,A -85,B 0,C 180,E1 17625.686,E2 17625.686} C_VEL
LIN {X 0,Y 442.858,Z 921.402,A -85,B 0,C 180,E1 17633.887,E2 17633.887} C_VEL
LIN {X 0,Y 440.99,Z 917.895,A -85,B 0,C 180,E1 17641.018,E2 17641.018} C_VEL
LIN {X 0,Y 445.487,Z 925.908,A -85,B 0,C 180,E1 17649.588,E2 17649.588} C_VEL
LIN {X 0,Y 456.842,Z 945.576,A -85,B 0,C 180,E1 17658.014,E2 17658.014} C_VEL
LIN {X 0,Y 472.215,Z 978.565,A -85,B 0,C 180,E1 17666.09,E2 17666.09} C_VEL
LIN {X 0,Y 481.93,Z 1010.377,A -85,B 0,C 180,E1 17671.385,E2 17671.385} C_VEL
LIN {X 0,Y 458.625,Z 1082.333,A -85,B 0,C 180,E1 17675.89,E2 17675.89} C_VEL
LIN {X 0,Y 432.982,Z 1144.515,A -85,B 0,C 180,E1 17682.276,E2 17682.276} C_VEL
LIN {X 0,Y 408.406,Z 1197.397,A -85,B 0,C 180,E1 17690.908,E2 17690.908} C_VEL
LIN {X 0,Y 390.361,Z 1238.021,A -85,B 0,C 180,E1 17701.582,E2 17701.582} C_VEL
LIN {X 0,Y 381.585,Z 1263.347,A -85,B 0,C 180,E1 17712.658,E2 17712.658} C_VEL
LIN {X 0,Y 379.333,Z 1274.675,A -85,B 0,C 180,E1 17721.957,E2 17721.957} C_VEL
LIN {X 0,Y 379.409,Z 1277.68,A -85,B 0,C 180,E1 17731.145,E2 17731.145} C_VEL
LIN {X 0,Y 379.834,Z 1271.145,A -85,B 0,C 180,E1 17741.718,E2 17741.718} C_VEL
LIN {X 0,Y 385.684,Z 1250.202,A -85,B 0,C 180,E1 17753.768,E2 17753.768} C_VEL
LIN {X 0,Y 400.075,Z 1215.035,A -85,B 0,C 180,E1 17765.029,E2 17765.029} C_VEL
LIN {X 0,Y 423.234,Z 1165.838,A -85,B 0,C 180,E1 17774.646,E2 17774.646} C_VEL
LIN {X 0,Y 449.472,Z 1105.918,A -85,B 0,C 180,E1 17781.94,E2 17781.94} C_VEL
LIN {X 0,Y 474.305,Z 1036.897,A -85,B 0,C 180,E1 17787.112,E2 17787.112} C_VEL
LIN {X 0,Y 481.906,Z 1006.627,A -85,B 0,C 180,E1 17788.89,E2 17788.89} C_VEL
LIN {X 0,Y 466.825,Z 965.542,A -85,B 0,C 180,E1 17796.509,E2 17796.509} C_VEL
LIN {X 0,Y 451.176,Z 934.833,A -85,B 0,C 180,E1 17805.453,E2 17805.453} C_VEL
LIN {X 0,Y 443.038,Z 921.528,A -85,B 0,C 180,E1 17813.085,E2 17813.085} C_VEL
LIN {X 0,Y 440.819,Z 917.125,A -85,B 0,C 180,E1 17820.461,E2 17820.461} C_VEL
LIN {X 0,Y 445.593,Z 925.895,A -85,B 0,C 180,E1 17829.645,E2 17829.645} C_VEL
LIN {X 0,Y 457.686,Z 946.457,A -85,B 0,C 180,E1 17838.236,E2 17838.236} C_VEL
LIN {X 0,Y 473.805,Z 980.783,A -85,B 0,C 180,E1 17846.342,E2 17846.342} C_VEL
LIN {X 0,Y 482.94,Z 1010.409,A -85,B 0,C 180,E1 17851.099,E2 17851.099} C_VEL
LIN {X 0,Y 460.402,Z 1082.345,A -85,B 0,C 180,E1 17855.412,E2 17855.412} C_VEL
LIN {X 0,Y 435.114,Z 1144.789,A -85,B 0,C 180,E1 17861.465,E2 17861.465} C_VEL
LIN {X 0,Y 410.454,Z 1198.571,A -85,B 0,C 180,E1 17869.715,E2 17869.715} C_VEL
LIN {X 0,Y 392.038,Z 1240.093,A -85,B 0,C 180,E1 17879.81,E2 17879.81} C_VEL
LIN {X 0,Y 382.038,Z 1268.626,A -85,B 0,C 180,E1 17891.164,E2 17891.164} C_VEL
LIN {X 0,Y 379.342,Z 1282.858,A -85,B 0,C 180,E1 17901.956,E2 17901.956} C_VEL
LIN {X 0,Y 378.845,Z 1285.982,A -85,B 0,C 180,E1 17911.147,E2 17911.147} C_VEL
LIN {X 0,Y 379.555,Z 1280.77,A -85,B 0,C 180,E1 17920.358,E2 17920.358} C_VEL
LIN {X 0,Y 383.38,Z 1263.773,A -85,B 0,C 180,E1 17931.294,E2 17931.294} C_VEL
LIN {X 0,Y 395.604,Z 1231.678,A -85,B 0,C 180,E1 17942.644,E2 17942.644} C_VEL
LIN {X 0,Y 417.101,Z 1184.515,A -85,B 0,C 180,E1 17952.818,E2 17952.818} C_VEL
LIN {X 0,Y 427.2,Z 1162.447,A -85,B 0,C 180,E1 17956.219,E2 17956.219} C_VEL
LIN {X 0,Y 431.545,Z 1140.395,A -85,B 0,C 180,E1 17959.888,E2 17959.888} C_VEL
LIN {X 0,Y 457.89,Z 1076.563,A -85,B 0,C 180,E1 17965.857,E2 17965.857} C_VEL
LIN {X 0,Y 478.086,Z 1010.271,A -85,B 0,C 180,E1 17969.907,E2 17969.907} C_VEL
LIN {X 0,Y 463.918,Z 971.944,A -85,B 0,C 180,E1 17977.183,E2 17977.183} C_VEL
LIN {X 0,Y 448.841,Z 942.215,A -85,B 0,C 180,E1 17986.16,E2 17986.16} C_VEL
LIN {X 0,Y 441.207,Z 929.148,A -85,B 0,C 180,E1 17994.021,E2 17994.021} C_VEL
LIN {X 0,Y 439.487,Z 925.881,A -85,B 0,C 180,E1 18001.268,E2 18001.268} C_VEL
LIN {X 0,Y 443.546,Z 933.71,A -85,B 0,C 180,E1 18009.513,E2 18009.513} C_VEL
LIN {X 0,Y 454.737,Z 953.916,A -85,B 0,C 180,E1 18018.168,E2 18018.168} C_VEL
LIN {X 0,Y 469.33,Z 987.55,A -85,B 0,C 180,E1 18026.262,E2 18026.262} C_VEL
LIN {X 0,Y 476.657,Z 1014.551,A -85,B 0,C 180,E1 18030.76,E2 18030.76} C_VEL
LIN {X 0,Y 452.501,Z 1085.987,A -85,B 0,C 180,E1 18035.341,E2 18035.341} C_VEL
LIN {X 0,Y 425.543,Z 1148.721,A -85,B 0,C 180,E1 18041.991,E2 18041.991} C_VEL
LIN {X 0,Y 400.646,Z 1200.195,A -85,B 0,C 180,E1 18050.723,E2 18050.723} C_VEL
LIN {X 0,Y 382.329,Z 1239.837,A -85,B 0,C 180,E1 18061.576,E2 18061.576} C_VEL
LIN {X 0,Y 373.514,Z 1264.213,A -85,B 0,C 180,E1 18072.768,E2 18072.768} C_VEL
LIN {X 0,Y 371.228,Z 1276.331,A -85,B 0,C 180,E1 18084.138,E2 18084.138} C_VEL
LIN {X 0,Y 371.199,Z 1277.309,A -85,B 0,C 180,E1 18093.514,E2 18093.514} C_VEL
LIN {X 0,Y 372.483,Z 1268.563,A -85,B 0,C 180,E1 18104.14,E2 18104.14} C_VEL
LIN {X 0,Y 379.194,Z 1246.77,A -85,B 0,C 180,E1 18115.737,E2 18115.737} C_VEL
LIN {X 0,Y 395.342,Z 1210.646,A -85,B 0,C 180,E1 18126.825,E2 18126.825} C_VEL
LIN {X 0,Y 419.768,Z 1160.54,A -85,B 0,C 180,E1 18136.26,E2 18136.26} C_VEL
LIN {X 0,Y 447.117,Z 1099.565,A -85,B 0,C 180,E1 18143.355,E2 18143.355} C_VEL
LIN {X 0,Y 471.972,Z 1029.791,A -85,B 0,C 180,E1 18148.375,E2 18148.375} C_VEL
LIN {X 0,Y 476.657,Z 1010.352,A -85,B 0,C 180,E1 18149.568,E2 18149.568} C_VEL
LIN {X 0,Y 462.461,Z 970.103,A -85,B 0,C 180,E1 18157.296,E2 18157.296} C_VEL
LIN {X 0,Y 448.158,Z 941.26,A -85,B 0,C 180,E1 18166.183,E2 18166.183} C_VEL
LIN {X 0,Y 441.248,Z 929.246,A -85,B 0,C 180,E1 18173.305,E2 18173.305} C_VEL
LIN {X 0,Y 439.305,Z 924.989,A -85,B 0,C 180,E1 18180.463,E2 18180.463} C_VEL
LIN {X 0,Y 443.709,Z 933.718,A -85,B 0,C 180,E1 18189.562,E2 18189.562} C_VEL
LIN {X 0,Y 455.269,Z 954.246,A -85,B 0,C 180,E1 18198.165,E2 18198.165} C_VEL
LIN {X 0,Y 470.638,Z 988.938,A -85,B 0,C 180,E1 18206.326,E2 18206.326} C_VEL
LIN {X 0,Y 477.789,Z 1013.826,A -85,B 0,C 180,E1 18210.428,E2 18210.428} C_VEL
LIN {X 0,Y 454.365,Z 1085.624,A -85,B 0,C 180,E1 18214.835,E2 18214.835} C_VEL
LIN {X 0,Y 428.219,Z 1147.695,A -85,B 0,C 180,E1 18221.015,E2 18221.015} C_VEL
LIN {X 0,Y 402.099,Z 1202.487,A -85,B 0,C 180,E1 18229.768,E2 18229.768} C_VEL
LIN {X 0,Y 383.189,Z 1243.546,A -85,B 0,C 180,E1 18240.349,E2 18240.349} C_VEL
LIN {X 0,Y 374.091,Z 1269.154,A -85,B 0,C 180,E1 18251.076,E2 18251.076} C_VEL
LIN {X 0,Y 371.355,Z 1282.77,A -85,B 0,C 180,E1 18261.782,E2 18261.782} C_VEL
LIN {X 0,Y 370.871,Z 1285.895,A -85,B 0,C 180,E1 18271.171,E2 18271.171} C_VEL
LIN {X 0,Y 371.569,Z 1280.682,A -85,B 0,C 180,E1 18280.583,E2 18280.583} C_VEL
LIN {X 0,Y 375.97,Z 1262.881,A -85,B 0,C 180,E1 18292.121,E2 18292.121} C_VEL
LIN {X 0,Y 389.625,Z 1229.487,A -85,B 0,C 180,E1 18303.871,E2 18303.871} C_VEL
LIN {X 0,Y 411.881,Z 1182.5,A -85,B 0,C 180,E1 18313.931,E2 18313.931} C_VEL
LIN {X 0,Y 431.545,Z 1140.395,A -85,B 0,C 180,E1 18319.888,E2 18319.888} C_VEL
LIN {X 0,Y 436.826,Z 1116.685,A -85,B 0,C 180,E1 18323.311,E2 18323.311} C_VEL
LIN {X 0,Y 463.453,Z 1048.017,A -85,B 0,C 180,E1 18328.599,E2 18328.599} C_VEL
LIN {X 0,Y 472.783,Z 1013.646,A -85,B 0,C 180,E1 18330.655,E2 18330.655} C_VEL
LIN {X 0,Y 459.123,Z 975.68,A -85,B 0,C 180,E1 18338.211,E2 18338.211} C_VEL
LIN {X 0,Y 445.555,Z 948.293,A -85,B 0,C 180,E1 18347.113,E2 18347.113} C_VEL
LIN {X 0,Y 439.01,Z 936.586,A -85,B 0,C 180,E1 18354.534,E2 18354.534} C_VEL
LIN {X 0,Y 437.723,Z 933.771,A -85,B 0,C 180,E1 18361.522,E2 18361.522} C_VEL
LIN {X 0,Y 441.722,Z 941.723,A -85,B 0,C 180,E1 18369.61,E2 18369.61} C_VEL
LIN {X 0,Y 452.122,Z 961.726,A -85,B 0,C 180,E1 18378.071,E2 18378.071} C_VEL
LIN {X 0,Y 465.616,Z 994.891,A -85,B 0,C 180,E1 18386.128,E2 18386.128} C_VEL
LIN {X 0,Y 471.383,Z 1018.866,A -85,B 0,C 180,E1 18390.123,E2 18390.123} C_VEL
LIN {X 0,Y 446.401,Z 1089.682,A -85,B 0,C 180,E1 18394.78,E2 18394.78} C_VEL
LIN {X 0,Y 418.219,Z 1152.611,A -85,B 0,C 180,E1 18401.651,E2 18401.651} C_VEL
LIN {X 0,Y 392.407,Z 1203.948,A -85,B 0,C 180,E1 18410.754,E2 18410.754} C_VEL
LIN {X 0,Y 373.627,Z 1243.175,A -85,B 0,C 180,E1 18422.175,E2 18422.175} C_VEL
LIN {X 0,Y 364.746,Z 1267.226,A -85,B 0,C 180,E1 18434.321,E2 18434.321} C_VEL
LIN {X 0,Y 363.221,Z 1276.419,A -85,B 0,C 180,E1 18444.009,E2 18444.009} C_VEL
LIN {X 0,Y 363.193,Z 1277.397,A -85,B 0,C 180,E1 18453.591,E2 18453.591} C_VEL
LIN {X 0,Y 364.563,Z 1268.653,A -85,B 0,C 180,E1 18464.454,E2 18464.454} C_VEL
LIN {X 0,Y 371.721,Z 1246.863,A -85,B 0,C 180,E1 18476.293,E2 18476.293} C_VEL
LIN {X 0,Y 388.609,Z 1210.81,A -85,B 0,C 180,E1 18487.552,E2 18487.552} C_VEL
LIN {X 0,Y 413.687,Z 1161.368,A -85,B 0,C 180,E1 18496.986,E2 18496.986} C_VEL
LIN {X 0,Y 441.805,Z 1100.706,A -85,B 0,C 180,E1 18504.117,E2 18504.117} C_VEL
LIN {X 0,Y 467.446,Z 1030.9,A -85,B 0,C 180,E1 18509.166,E2 18509.166} C_VEL
LIN {X 0,Y 471.392,Z 1013.806,A -85,B 0,C 180,E1 18510.309,E2 18510.309} C_VEL
LIN {X 0,Y 458.946,Z 976.753,A -85,B 0,C 180,E1 18517.625,E2 18517.625} C_VEL
LIN {X 0,Y 445.61,Z 948.406,A -85,B 0,C 180,E1 18526.551,E2 18526.551} C_VEL
LIN {X 0,Y 439.222,Z 936.866,A -85,B 0,C 180,E1 18533.523,E2 18533.523} C_VEL
LIN {X 0,Y 437.568,Z 932.797,A -85,B 0,C 180,E1 18540.464,E2 18540.464} C_VEL
LIN {X 0,Y 441.955,Z 941.825,A -85,B 0,C 180,E1 18549.725,E2 18549.725} C_VEL
LIN {X 0,Y 452.731,Z 962.317,A -85,B 0,C 180,E1 18558.132,E2 18558.132} C_VEL
LIN {X 0,Y 466.562,Z 995.3,A -85,B 0,C 180,E1 18566.003,E2 18566.003} C_VEL
LIN {X 0,Y 472.407,Z 1018.237,A -85,B 0,C 180,E1 18569.787,E2 18569.787} C_VEL
LIN {X 0,Y 447.768,Z 1090.372,A -85,B 0,C 180,E1 18574.355,E2 18574.355} C_VEL
LIN {X 0,Y 420.551,Z 1152.267,A -85,B 0,C 180,E1 18580.764,E2 18580.764} C_VEL
LIN {X 0,Y 394.364,Z 1205.066,A -85,B 0,C 180,E1 18589.539,E2 18589.539} C_VEL
LIN {X 0,Y 375.178,Z 1245.175,A -85,B 0,C 180,E1 18600.307,E2 18600.307} C_VEL
LIN {X 0,Y 365.817,Z 1271.057,A -85,B 0,C 180,E1 18611.885,E2 18611.885} C_VEL
LIN {X 0,Y 363.37,Z 1282.681,A -85,B 0,C 180,E1 18621.6,E2 18621.6} C_VEL
LIN {X 0,Y 362.872,Z 1285.807,A -85,B 0,C 180,E1 18631.197,E2 18631.197} C_VEL
LIN {X 0,Y 363.712,Z 1279.781,A -85,B 0,C 180,E1 18641.622,E2 18641.622} C_VEL
LIN {X 0,Y 368.647,Z 1261.904,A -85,B 0,C 180,E1 18653.005,E2 18653.005} C_VEL
LIN {X 0,Y 383.476,Z 1227.81,A -85,B 0,C 180,E1 18664.99,E2 18664.99} C_VEL
LIN {X 0,Y 406.976,Z 1180.206,A -85,B 0,C 180,E1 18675.115,E2 18675.115} C_VEL
LIN {X 0,Y 435.013,Z 1120.812,A -85,B 0,C 180,E1 18682.888,E2 18682.888} C_VEL
LIN {X 0,Y 436.826,Z 1116.685,A -85,B 0,C 180,E1 18683.311,E2 18683.311} C_VEL
LIN {X 0,Y 442.795,Z 1091.36,A -85,B 0,C 180,E1 18686.451,E2 18686.451} C_VEL
LIN {X 0,Y 468.078,Z 1019.091,A -85,B 0,C 180,E1 18691.074,E2 18691.074} C_VEL
LIN {X 0,Y 455.622,Z 982.341,A -85,B 0,C 180,E1 18698.548,E2 18698.548} C_VEL
LIN {X 0,Y 442.847,Z 955.387,A -85,B 0,C 180,E1 18707.469,E2 18707.469} C_VEL
LIN {X 0,Y 436.996,Z 944.196,A -85,B 0,C 180,E1 18714.781,E2 18714.781} C_VEL
LIN {X 0,Y 435.861,Z 941.539,A -85,B 0,C 180,E1 18721.528,E2 18721.528} C_VEL
LIN {X 0,Y 439.83,Z 949.738,A -85,B 0,C 180,E1 18729.767,E2 18729.767} C_VEL
LIN {X 0,Y 449.645,Z 970.315,A -85,B 0,C 180,E1 18738.218,E2 18738.218} C_VEL
LIN {X 0,Y 462.048,Z 1002.723,A -85,B 0,C 180,E1 18746.083,E2 18746.083} C_VEL
LIN {X 0,Y 466.062,Z 1023.231,A -85,B 0,C 180,E1 18749.48,E2 18749.48} C_VEL
LIN {X 0,Y 440.196,Z 1093.48,A -85,B 0,C 180,E1 18754.227,E2 18754.227} C_VEL
LIN {X 0,Y 411.954,Z 1154.185,A -85,B 0,C 180,E1 18761.004,E2 18761.004} C_VEL
LIN {X 0,Y 385.418,Z 1204.98,A -85,B 0,C 180,E1 18770.19,E2 18770.19} C_VEL
LIN {X 0,Y 366.264,Z 1243.264,A -85,B 0,C 180,E1 18781.565,E2 18781.565} C_VEL
LIN {X 0,Y 356.894,Z 1267.315,A -85,B 0,C 180,E1 18793.966,E2 18793.966} C_VEL
LIN {X 0,Y 355.215,Z 1276.507,A -85,B 0,C 180,E1 18803.873,E2 18803.873} C_VEL
LIN {X 0,Y 355.209,Z 1277.485,A -85,B 0,C 180,E1 18813.672,E2 18813.672} C_VEL
LIN {X 0,Y 356.676,Z 1268.743,A -85,B 0,C 180,E1 18824.78,E2 18824.78} C_VEL
LIN {X 0,Y 364.017,Z 1247.613,A -85,B 0,C 180,E1 18836.605,E2 18836.605} C_VEL
LIN {X 0,Y 381.437,Z 1212.03,A -85,B 0,C 180,E1 18848.043,E2 18848.043} C_VEL
LIN {X 0,Y 406.905,Z 1163.763,A -85,B 0,C 180,E1 18857.496,E2 18857.496} C_VEL
LIN {X 0,Y 435.599,Z 1104.154,A -85,B 0,C 180,E1 18864.684,E2 18864.684} C_VEL
LIN {X 0,Y 461.996,Z 1035.311,A -85,B 0,C 180,E1 18869.783,E2 18869.783} C_VEL
LIN {X 0,Y 466.688,Z 1019.229,A -85,B 0,C 180,E1 18870.737,E2 18870.737} C_VEL
LIN {X 0,Y 454.879,Z 982.29,A -85,B 0,C 180,E1 18878.268,E2 18878.268} C_VEL
LIN {X 0,Y 442.654,Z 955.117,A -85,B 0,C 180,E1 18887.096,E2 18887.096} C_VEL
LIN {X 0,Y 437.035,Z 944.357,A -85,B 0,C 180,E1 18893.99,E2 18893.99} C_VEL
LIN {X 0,Y 435.705,Z 940.565,A -85,B 0,C 180,E1 18900.466,E2 18900.466} C_VEL
LIN {X 0,Y 439.902,Z 949.576,A -85,B 0,C 180,E1 18909.646,E2 18909.646} C_VEL
LIN {X 0,Y 449.539,Z 968.7,A -85,B 0,C 180,E1 18917.648,E2 18917.648} C_VEL
LIN {X 0,Y 462.307,Z 1001.105,A -85,B 0,C 180,E1 18925.564,E2 18925.564} C_VEL
LIN {X 0,Y 467.198,Z 1022.431,A -85,B 0,C 180,E1 18929.132,E2 18929.132} C_VEL
LIN {X 0,Y 442.08,Z 1093.073,A -85,B 0,C 180,E1 18933.707,E2 18933.707} C_VEL
LIN {X 0,Y 413.881,Z 1154.817,A -85,B 0,C 180,E1 18940.241,E2 18940.241} C_VEL
LIN {X 0,Y 386.651,Z 1207.645,A -85,B 0,C 180,E1 18949.302,E2 18949.302} C_VEL
LIN {X 0,Y 367.193,Z 1246.766,A -85,B 0,C 180,E1 18960.251,E2 18960.251} C_VEL
LIN {X 0,Y 357.635,Z 1272.563,A -85,B 0,C 180,E1 18972.502,E2 18972.502} C_VEL
LIN {X 0,Y 355.151,Z 1284.213,A -85,B 0,C 180,E1 18983.872,E2 18983.872} C_VEL
LIN {X 0,Y 355.135,Z 1285.262,A -85,B 0,C 180,E1 18993.672,E2 18993.672} C_VEL
LIN {X 0,Y 356.502,Z 1276.35,A -85,B 0,C 180,E1 19004.787,E2 19004.787} C_VEL
LIN {X 0,Y 364.684,Z 1253.028,A -85,B 0,C 180,E1 19017.341,E2 19017.341} C_VEL
LIN {X 0,Y 382.69,Z 1215.336,A -85,B 0,C 180,E1 19028.926,E2 19028.926} C_VEL
LIN {X 0,Y 409.072,Z 1164.498,A -85,B 0,C 180,E1 19038.408,E2 19038.408} C_VEL
LIN {X 0,Y 438.039,Z 1102.43,A -85,B 0,C 180,E1 19045.529,E2 19045.529} C_VEL
LIN {X 0,Y 442.795,Z 1091.36,A -85,B 0,C 180,E1 19046.451,E2 19046.451} C_VEL
LIN {X 0,Y 449.161,Z 1064.44,A -85,B 0,C 180,E1 19049.312,E2 19049.312} C_VEL
LIN {X 0,Y 462.797,Z 1022.068,A -85,B 0,C 180,E1 19051.922,E2 19051.922} C_VEL
LIN {X 0,Y 451.369,Z 987.117,A -85,B 0,C 180,E1 19059.369,E2 19059.369} C_VEL
LIN {X 0,Y 439.558,Z 961.189,A -85,B 0,C 180,E1 19068.416,E2 19068.416} C_VEL
LIN {X 0,Y 434.601,Z 951.39,A -85,B 0,C 180,E1 19075.528,E2 19075.528} C_VEL
LIN {X 0,Y 433.986,Z 949.412,A -85,B 0,C 180,E1 19082.036,E2 19082.036} C_VEL
LIN {X 0,Y 438.64,Z 958.938,A -85,B 0,C 180,E1 19090.862,E2 19090.862} C_VEL
LIN {X 0,Y 449.878,Z 985.162,A -85,B 0,C 180,E1 19100.271,E2 19100.271} C_VEL
LIN {X 0,Y 461.233,Z 1021.988,A -85,B 0,C 180,E1 19108.224,E2 19108.224} C_VEL
LIN {X 0,Y 457.672,Z 1037.026,A -85,B 0,C 180,E1 19109.361,E2 19109.361} C_VEL
LIN {X 0,Y 431.191,Z 1103.646,A -85,B 0,C 180,E1 19114.258,E2 19114.258} C_VEL
LIN {X 0,Y 401.261,Z 1164.197,A -85,B 0,C 180,E1 19121.587,E2 19121.587} C_VEL
LIN {X 0,Y 375.024,Z 1212.45,A -85,B 0,C 180,E1 19131.186,E2 19131.186} C_VEL
LIN {X 0,Y 356.816,Z 1247.923,A -85,B 0,C 180,E1 19142.813,E2 19142.813} C_VEL
LIN {X 0,Y 348.58,Z 1268.952,A -85,B 0,C 180,E1 19154.869,E2 19154.869} C_VEL
LIN {X 0,Y 347.057,Z 1277.614,A -85,B 0,C 180,E1 19166.242,E2 19166.242} C_VEL
LIN {X 0,Y 347.279,Z 1276.554,A -85,B 0,C 180,E1 19176.268,E2 19176.268} C_VEL
LIN {X 0,Y 349.83,Z 1264.656,A -85,B 0,C 180,E1 19188.222,E2 19188.222} C_VEL
LIN {X 0,Y 360.062,Z 1240.293,A -85,B 0,C 180,E1 19200.186,E2 19200.186} C_VEL
LIN {X 0,Y 380.977,Z 1201.207,A -85,B 0,C 180,E1 19211.421,E2 19211.421} C_VEL
LIN {X 0,Y 409.111,Z 1148.963,A -85,B 0,C 180,E1 19220.528,E2 19220.528} C_VEL
LIN {X 0,Y 438.227,Z 1087.504,A -85,B 0,C 180,E1 19227.056,E2 19227.056} C_VEL
LIN {X 0,Y 461.485,Z 1022.736,A -85,B 0,C 180,E1 19231.498,E2 19231.498} C_VEL
LIN {X 0,Y 450.294,Z 986.442,A -85,B 0,C 180,E1 19239.25,E2 19239.25} C_VEL
LIN {X 0,Y 438.752,Z 958.612,A -85,B 0,C 180,E1 19248.882,E2 19248.882} C_VEL
LIN {X 0,Y 433.995,Z 947.728,A -85,B 0,C 180,E1 19258.966,E2 19258.966} C_VEL
LIN {X 0,Y 437.362,Z 956.831,A -85,B 0,C 180,E1 19269.325,E2 19269.325} C_VEL
LIN {X 0,Y 446.843,Z 977.088,A -85,B 0,C 180,E1 19277.758,E2 19277.758} C_VEL
LIN {X 0,Y 458.587,Z 1008.43,A -85,B 0,C 180,E1 19285.436,E2 19285.436} C_VEL
LIN {X 0,Y 461.895,Z 1026.967,A -85,B 0,C 180,E1 19288.475,E2 19288.475} C_VEL
LIN {X 0,Y 435.246,Z 1098.384,A -85,B 0,C 180,E1 19293.255,E2 19293.255} C_VEL
LIN {X 0,Y 406.011,Z 1159.724,A -85,B 0,C 180,E1 19300.029,E2 19300.029} C_VEL
LIN {X 0,Y 378.65,Z 1210.706,A -85,B 0,C 180,E1 19309.186,E2 19309.186} C_VEL
LIN {X 0,Y 359.063,Z 1248.678,A -85,B 0,C 180,E1 19320.31,E2 19320.31} C_VEL
LIN {X 0,Y 349.5,Z 1273.624,A -85,B 0,C 180,E1 19332.851,E2 19332.851} C_VEL
LIN {X 0,Y 347.149,Z 1284.125,A -85,B 0,C 180,E1 19343.73,E2 19343.73} C_VEL
LIN {X 0,Y 347.125,Z 1285.174,A -85,B 0,C 180,E1 19353.757,E2 19353.757} C_VEL
LIN {X 0,Y 348.607,Z 1276.261,A -85,B 0,C 180,E1 19365.13,E2 19365.13} C_VEL
LIN {X 0,Y 357.103,Z 1253.214,A -85,B 0,C 180,E1 19377.849,E2 19377.849} C_VEL
LIN {X 0,Y 375.964,Z 1215.594,A -85,B 0,C 180,E1 19389.651,E2 19389.651} C_VEL
LIN {X 0,Y 403.257,Z 1165.051,A -85,B 0,C 180,E1 19399.197,E2 19399.197} C_VEL
LIN {X 0,Y 432.861,Z 1103.614,A -85,B 0,C 180,E1 19406.313,E2 19406.313} C_VEL
LIN {X 0,Y 449.161,Z 1064.44,A -85,B 0,C 180,E1 19409.312,E2 19409.312} C_VEL
LIN {X 0,Y 455.195,Z 1036.086,A -85,B 0,C 180,E1 19411.907,E2 19411.907} C_VEL
LIN {X 0,Y 457.574,Z 1025.176,A -85,B 0,C 180,E1 19412.784,E2 19412.784} C_VEL
LIN {X 0,Y 446.967,Z 991.757,A -85,B 0,C 180,E1 19420.234,E2 19420.234} C_VEL
LIN {X 0,Y 436.105,Z 966.089,A -85,B 0,C 180,E1 19429.763,E2 19429.763} C_VEL
LIN {X 0,Y 431.883,Z 956.194,A -85,B 0,C 180,E1 19439.026,E2 19439.026} C_VEL
LIN {X 0,Y 434.602,Z 964.031,A -85,B 0,C 180,E1 19448.911,E2 19448.911} C_VEL
LIN {X 0,Y 443.097,Z 983.797,A -85,B 0,C 180,E1 19457.506,E2 19457.506} C_VEL
LIN {X 0,Y 453.623,Z 1015.706,A -85,B 0,C 180,E1 19465.538,E2 19465.538} C_VEL
LIN {X 0,Y 455.691,Z 1031.096,A -85,B 0,C 180,E1 19468.126,E2 19468.126} C_VEL
LIN {X 0,Y 428.272,Z 1100.013,A -85,B 0,C 180,E1 19473,E2 19473} C_VEL
LIN {X 0,Y 397.659,Z 1160.817,A -85,B 0,C 180,E1 19480.166,E2 19480.166} C_VEL
LIN {X 0,Y 369.815,Z 1210.155,A -85,B 0,C 180,E1 19489.771,E2 19489.771} C_VEL
LIN {X 0,Y 350.154,Z 1246.49,A -85,B 0,C 180,E1 19501.549,E2 19501.549} C_VEL
LIN {X 0,Y 341.241,Z 1267.492,A -85,B 0,C 180,E1 19513.21,E2 19513.21} C_VEL
LIN {X 0,Y 339.217,Z 1276.683,A -85,B 0,C 180,E1 19523.583,E2 19523.583} C_VEL
LIN {X 0,Y 339.215,Z 1277.661,A -85,B 0,C 180,E1 19533.845,E2 19533.845} C_VEL
LIN {X 0,Y 340.86,Z 1268.924,A -85,B 0,C 180,E1 19545.483,E2 19545.483} C_VEL
LIN {X 0,Y 349.168,Z 1247.796,A -85,B 0,C 180,E1 19557.834,E2 19557.834} C_VEL
LIN {X 0,Y 368.395,Z 1212.218,A -85,B 0,C 180,E1 19569.648,E2 19569.648} C_VEL
LIN {X 0,Y 396.178,Z 1163.332,A -85,B 0,C 180,E1 19579.366,E2 19579.366} C_VEL
LIN {X 0,Y 426.853,Z 1103.082,A -85,B 0,C 180,E1 19586.607,E2 19586.607} C_VEL
LIN {X 0,Y 454.737,Z 1033.228,A -85,B 0,C 180,E1 19591.693,E2 19591.693} C_VEL
LIN {X 0,Y 455.936,Z 1024.582,A -85,B 0,C 180,E1 19592.575,E2 19592.575} C_VEL
LIN {X 0,Y 445.263,Z 989.263,A -85,B 0,C 180,E1 19600.624,E2 19600.624} C_VEL
LIN {X 0,Y 435.389,Z 964.785,A -85,B 0,C 180,E1 19609.997,E2 19609.997} C_VEL
LIN {X 0,Y 431.679,Z 955.641,A -85,B 0,C 180,E1 19619.464,E2 19619.464} C_VEL
LIN {X 0,Y 435.076,Z 964.594,A -85,B 0,C 180,E1 19629.311,E2 19629.311} C_VEL
LIN {X 0,Y 444.415,Z 985.877,A -85,B 0,C 180,E1 19638.032,E2 19638.032} C_VEL
LIN {X 0,Y 455.381,Z 1018.555,A -85,B 0,C 180,E1 19645.893,E2 19645.893} C_VEL
LIN {X 0,Y 457.148,Z 1029.581,A -85,B 0,C 180,E1 19647.722,E2 19647.722} C_VEL
LIN {X 0,Y 430.092,Z 1099.756,A -85,B 0,C 180,E1 19652.466,E2 19652.466} C_VEL
LIN {X 0,Y 400.047,Z 1160.774,A -85,B 0,C 180,E1 19659.28,E2 19659.28} C_VEL
LIN {X 0,Y 371.513,Z 1211.995,A -85,B 0,C 180,E1 19668.674,E2 19668.674} C_VEL
LIN {X 0,Y 351.09,Z 1250,A -85,B 0,C 180,E1 19680.215,E2 19680.215} C_VEL
LIN {X 0,Y 341.295,Z 1274.579,A -85,B 0,C 180,E1 19693.212,E2 19693.212} C_VEL
LIN {X 0,Y 339.147,Z 1284.037,A -85,B 0,C 180,E1 19703.581,E2 19703.581} C_VEL
LIN {X 0,Y 339.13,Z 1285.087,A -85,B 0,C 180,E1 19713.846,E2 19713.846} C_VEL
LIN {X 0,Y 340.726,Z 1276.172,A -85,B 0,C 180,E1 19725.489,E2 19725.489} C_VEL
LIN {X 0,Y 349.687,Z 1253.123,A -85,B 0,C 180,E1 19738.493,E2 19738.493} C_VEL
LIN {X 0,Y 369.684,Z 1215.176,A -85,B 0,C 180,E1 19750.567,E2 19750.567} C_VEL
LIN {X 0,Y 398.171,Z 1164.332,A -85,B 0,C 180,E1 19760.205,E2 19760.205} C_VEL
LIN {X 0,Y 428.848,Z 1102.434,A -85,B 0,C 180,E1 19767.328,E2 19767.328} C_VEL
LIN {X 0,Y 455.195,Z 1036.086,A -85,B 0,C 180,E1 19771.907,E2 19771.907} C_VEL
LIN {X 0,Y 454.582,Z 1029.025,A -85,B 0,C 180,E1 19773.01,E2 19773.01} C_VEL
LIN {X 0,Y 451.307,Z 1024.124,A -85,B 0,C 180,E1 19774.491,E2 19774.491} C_VEL
LIN {X 0,Y 440.99,Z 992.55,A -85,B 0,C 180,E1 19782.361,E2 19782.361} C_VEL
LIN {X 0,Y 432.549,Z 972.174,A -85,B 0,C 180,E1 19790.952,E2 19790.952} C_VEL
LIN {X 0,Y 429.479,Z 964.276,A -85,B 0,C 180,E1 19800.539,E2 19800.539} C_VEL
LIN {X 0,Y 432.231,Z 972.024,A -85,B 0,C 180,E1 19809.12,E2 19809.12} C_VEL
LIN {X 0,Y 440.128,Z 991.94,A -85,B 0,C 180,E1 19817.628,E2 19817.628} C_VEL
LIN {X 0,Y 449.731,Z 1023.636,A -85,B 0,C 180,E1 19825.566,E2 19825.566} C_VEL
LIN {X 0,Y 450.522,Z 1035.294,A -85,B 0,C 180,E1 19827.442,E2 19827.442} C_VEL
LIN {X 0,Y 422.659,Z 1102.667,A -85,B 0,C 180,E1 19832.302,E2 19832.302} C_VEL
LIN {X 0,Y 391.322,Z 1162.746,A -85,B 0,C 180,E1 19839.516,E2 19839.516} C_VEL
LIN {X 0,Y 362.762,Z 1211.437,A -85,B 0,C 180,E1 19849.217,E2 19849.217} C_VEL
LIN {X 0,Y 342.092,Z 1248.102,A -85,B 0,C 180,E1 19861.539,E2 19861.539} C_VEL
LIN {X 0,Y 332.835,Z 1269.129,A -85,B 0,C 180,E1 19874.134,E2 19874.134} C_VEL
LIN {X 0,Y 331.078,Z 1277.789,A -85,B 0,C 180,E1 19886.06,E2 19886.06} C_VEL
LIN {X 0,Y 331.279,Z 1276.731,A -85,B 0,C 180,E1 19896.572,E2 19896.572} C_VEL
LIN {X 0,Y 333.971,Z 1265.651,A -85,B 0,C 180,E1 19908.534,E2 19908.534} C_VEL
LIN {X 0,Y 345.303,Z 1241.417,A -85,B 0,C 180,E1 19921.22,E2 19921.22} C_VEL
LIN {X 0,Y 367.884,Z 1202.662,A -85,B 0,C 180,E1 19932.858,E2 19932.858} C_VEL
LIN {X 0,Y 397.812,Z 1150.921,A -85,B 0,C 180,E1 19942.135,E2 19942.135} C_VEL
LIN {X 0,Y 428.922,Z 1089.081,A -85,B 0,C 180,E1 19948.782,E2 19948.782} C_VEL
LIN {X 0,Y 451.208,Z 1030.203,A -85,B 0,C 180,E1 19952.971,E2 19952.971} C_VEL
LIN {X 0,Y 441.683,Z 996.033,A -85,B 0,C 180,E1 19960.922,E2 19960.922} C_VEL
LIN {X 0,Y 432.911,Z 972.691,A -85,B 0,C 180,E1 19969.876,E2 19969.876} C_VEL
LIN {X 0,Y 429.408,Z 963.502,A -85,B 0,C 180,E1 19979.967,E2 19979.967} C_VEL
LIN {X 0,Y 432.413,Z 971.894,A -85,B 0,C 180,E1 19989.05,E2 19989.05} C_VEL
LIN {X 0,Y 440.78,Z 992.234,A -85,B 0,C 180,E1 19997.58,E2 19997.58} C_VEL
LIN {X 0,Y 451.012,Z 1024.598,A -85,B 0,C 180,E1 20005.532,E2 20005.532} C_VEL
LIN {X 0,Y 451.503,Z 1035.109,A -85,B 0,C 180,E1 20007.114,E2 20007.114} C_VEL
LIN {X 0,Y 422.687,Z 1106.106,A -85,B 0,C 180,E1 20012.1,E2 20012.1} C_VEL
LIN {X 0,Y 391.569,Z 1166.517,A -85,B 0,C 180,E1 20019.213,E2 20019.213} C_VEL
LIN {X 0,Y 361.969,Z 1217.43,A -85,B 0,C 180,E1 20029.166,E2 20029.166} C_VEL
LIN {X 0,Y 341.612,Z 1254.555,A -85,B 0,C 180,E1 20041.495,E2 20041.495} C_VEL
LIN {X 0,Y 332.891,Z 1276.073,A -85,B 0,C 180,E1 20054.137,E2 20054.137} C_VEL
LIN {X 0,Y 331.169,Z 1284.996,A -85,B 0,C 180,E1 20066.061,E2 20066.061} C_VEL
LIN {X 0,Y 331.148,Z 1283.952,A -85,B 0,C 180,E1 20076.574,E2 20076.574} C_VEL
LIN {X 0,Y 334.024,Z 1272.657,A -85,B 0,C 180,E1 20088.531,E2 20088.531} C_VEL
LIN {X 0,Y 344.725,Z 1248.157,A -85,B 0,C 180,E1 20101.214,E2 20101.214} C_VEL
LIN {X 0,Y 367.13,Z 1208.756,A -85,B 0,C 180,E1 20112.967,E2 20112.967} C_VEL
LIN {X 0,Y 397.397,Z 1156.036,A -85,B 0,C 180,E1 20122.33,E2 20122.33} C_VEL
LIN {X 0,Y 428.271,Z 1094.341,A -85,B 0,C 180,E1 20128.931,E2 20128.931} C_VEL
LIN {X 0,Y 452.628,Z 1029.689,A -85,B 0,C 180,E1 20133.392,E2 20133.392} C_VEL
LIN {X 0,Y 451.307,Z 1024.124,A -85,B 0,C 180,E1 20134.491,E2 20134.491} C_VEL
LIN {X 0,Y 442.226,Z 1013.206,A -85,B 0,C 180,E1 20138.691,E2 20138.691} C_VEL
LIN {X 0,Y 432.438,Z 985.651,A -85,B 0,C 180,E1 20147.812,E2 20147.812} C_VEL
LIN {X 0,Y 427.84,Z 974.807,A -85,B 0,C 180,E1 20154.947,E2 20154.947} C_VEL
LIN {X 0,Y 427.021,Z 972.079,A -85,B 0,C 180,E1 20161.051,E2 20161.051} C_VEL
LIN {X 0,Y 430.389,Z 981.298,A -85,B 0,C 180,E1 20170.184,E2 20170.184} C_VEL
LIN {X 0,Y 438.767,Z 1004.84,A -85,B 0,C 180,E1 20179.209,E2 20179.209} C_VEL
LIN {X 0,Y 446.474,Z 1036.044,A -85,B 0,C 180,E1 20186.519,E2 20186.519} C_VEL
LIN {X 0,Y 417.226,Z 1105.041,A -85,B 0,C 180,E1 20191.556,E2 20191.556} C_VEL
LIN {X 0,Y 384.706,Z 1165.241,A -85,B 0,C 180,E1 20198.929,E2 20198.929} C_VEL
LIN {X 0,Y 355.031,Z 1213.914,A -85,B 0,C 180,E1 20208.947,E2 20208.947} C_VEL
LIN {X 0,Y 334.038,Z 1249.703,A -85,B 0,C 180,E1 20221.53,E2 20221.53} C_VEL
LIN {X 0,Y 324.498,Z 1270.767,A -85,B 0,C 180,E1 20235.106,E2 20235.106} C_VEL
LIN {X 0,Y 323.072,Z 1277.876,A -85,B 0,C 180,E1 20245.963,E2 20245.963} C_VEL
LIN {X 0,Y 323.297,Z 1276.819,A -85,B 0,C 180,E1 20256.735,E2 20256.735} C_VEL
LIN {X 0,Y 326.19,Z 1265.742,A -85,B 0,C 180,E1 20268.993,E2 20268.993} C_VEL
LIN {X 0,Y 338.309,Z 1241.366,A -85,B 0,C 180,E1 20282.003,E2 20282.003} C_VEL
LIN {X 0,Y 362.758,Z 1201.156,A -85,B 0,C 180,E1 20294.117,E2 20294.117} C_VEL
LIN {X 0,Y 394.338,Z 1148.204,A -85,B 0,C 180,E1 20303.463,E2 20303.463} C_VEL
LIN {X 0,Y 425.601,Z 1087.212,A -85,B 0,C 180,E1 20309.885,E2 20309.885} C_VEL
LIN {X 0,Y 446.151,Z 1034.005,A -85,B 0,C 180,E1 20313.732,E2 20313.732} C_VEL
LIN {X 0,Y 437.596,Z 1001.177,A -85,B 0,C 180,E1 20321.696,E2 20321.696} C_VEL
LIN {X 0,Y 429.623,Z 978.835,A -85,B 0,C 180,E1 20330.824,E2 20330.824} C_VEL
LIN {X 0,Y 427.181,Z 970.74,A -85,B 0,C 180,E1 20338.95,E2 20338.95} C_VEL
LIN {X 0,Y 429.847,Z 979.582,A -85,B 0,C 180,E1 20349.105,E2 20349.105} C_VEL
LIN {X 0,Y 438.264,Z 1001.666,A -85,B 0,C 180,E1 20358.117,E2 20358.117} C_VEL
LIN {X 0,Y 447.367,Z 1035.001,A -85,B 0,C 180,E1 20366.061,E2 20366.061} C_VEL
LIN {X 0,Y 418.235,Z 1106.3,A -85,B 0,C 180,E1 20371.171,E2 20371.171} C_VEL
LIN {X 0,Y 386.297,Z 1166.497,A -85,B 0,C 180,E1 20378.264,E2 20378.264} C_VEL
LIN {X 0,Y 355.869,Z 1216.963,A -85,B 0,C 180,E1 20388.186,E2 20388.186} C_VEL
LIN {X 0,Y 335.015,Z 1252.913,A -85,B 0,C 180,E1 20400.136,E2 20400.136} C_VEL
LIN {X 0,Y 324.993,Z 1276.149,A -85,B 0,C 180,E1 20413.886,E2 20413.886} C_VEL
LIN {X 0,Y 323.154,Z 1284.908,A -85,B 0,C 180,E1 20425.963,E2 20425.963} C_VEL
LIN {X 0,Y 323.149,Z 1283.864,A -85,B 0,C 180,E1 20436.738,E2 20436.738} C_VEL
LIN {X 0,Y 326.199,Z 1272.567,A -85,B 0,C 180,E1 20448.992,E2 20448.992} C_VEL
LIN {X 0,Y 337.747,Z 1247.79,A -85,B 0,C 180,E1 20462.054,E2 20462.054} C_VEL
LIN {X 0,Y 361.029,Z 1208.666,A -85,B 0,C 180,E1 20473.876,E2 20473.876} C_VEL
LIN {X 0,Y 392.411,Z 1155.834,A -85,B 0,C 180,E1 20483.31,E2 20483.31} C_VEL
LIN {X 0,Y 424.411,Z 1093.497,A -85,B 0,C 180,E1 20489.945,E2 20489.945} C_VEL
LIN {X 0,Y 447.608,Z 1033.852,A -85,B 0,C 180,E1 20494.081,E2 20494.081} C_VEL
LIN {X 0,Y 442.226,Z 1013.206,A -85,B 0,C 180,E1 20498.691,E2 20498.691} C_VEL
LIN {X 0,Y 433.808,Z 1005.675,A -85,B 0,C 180,E1 20503.12,E2 20503.12} C_VEL
LIN {X 0,Y 426.914,Z 986.498,A -85,B 0,C 180,E1 20511.577,E2 20511.577} C_VEL
LIN {X 0,Y 424.686,Z 979.113,A -85,B 0,C 180,E1 20519.01,E2 20519.01} C_VEL
LIN {X 0,Y 426.996,Z 987.44,A -85,B 0,C 180,E1 20529.233,E2 20529.233} C_VEL
LIN {X 0,Y 433.856,Z 1008.04,A -85,B 0,C 180,E1 20537.85,E2 20537.85} C_VEL
LIN {X 0,Y 441.486,Z 1039.802,A -85,B 0,C 180,E1 20545.745,E2 20545.745} C_VEL
LIN {X 0,Y 410.784,Z 1109.56,A -85,B 0,C 180,E1 20551.009,E2 20551.009} C_VEL
LIN {X 0,Y 377.616,Z 1168.436,A -85,B 0,C 180,E1 20558.452,E2 20558.452} C_VEL
LIN {X 0,Y 347.327,Z 1216.213,A -85,B 0,C 180,E1 20568.67,E2 20568.67} C_VEL
LIN {X 0,Y 325.868,Z 1251.235,A -85,B 0,C 180,E1 20581.572,E2 20581.572} C_VEL
LIN {X 0,Y 316.651,Z 1270.855,A -85,B 0,C 180,E1 20594.728,E2 20594.728} C_VEL
LIN {X 0,Y 315.067,Z 1277.964,A -85,B 0,C 180,E1 20605.86,E2 20605.86} C_VEL
LIN {X 0,Y 315.296,Z 1276.908,A -85,B 0,C 180,E1 20616.907,E2 20616.907} C_VEL
LIN {X 0,Y 318.43,Z 1265.833,A -85,B 0,C 180,E1 20629.474,E2 20629.474} C_VEL
LIN {X 0,Y 330.997,Z 1241.958,A -85,B 0,C 180,E1 20642.572,E2 20642.572} C_VEL
LIN {X 0,Y 356.495,Z 1201.734,A -85,B 0,C 180,E1 20654.944,E2 20654.944} C_VEL
LIN {X 0,Y 388.583,Z 1149.845,A -85,B 0,C 180,E1 20664.236,E2 20664.236} C_VEL
LIN {X 0,Y 420.754,Z 1089.035,A -85,B 0,C 180,E1 20670.713,E2 20670.713} C_VEL
LIN {X 0,Y 441.417,Z 1039.305,A -85,B 0,C 180,E1 20674.217,E2 20674.217} C_VEL
LIN {X 0,Y 433.748,Z 1007.412,A -85,B 0,C 180,E1 20682.146,E2 20682.146} C_VEL
LIN {X 0,Y 426.99,Z 986.58,A -85,B 0,C 180,E1 20690.767,E2 20690.767} C_VEL
LIN {X 0,Y 424.597,Z 978.388,A -85,B 0,C 180,E1 20698.943,E2 20698.943} C_VEL
LIN {X 0,Y 427.255,Z 987.307,A -85,B 0,C 180,E1 20709.161,E2 20709.161} C_VEL
LIN {X 0,Y 435.006,Z 1009.702,A -85,B 0,C 180,E1 20718.196,E2 20718.196} C_VEL
LIN {X 0,Y 442.511,Z 1039.742,A -85,B 0,C 180,E1 20725.475,E2 20725.475} C_VEL
LIN {X 0,Y 412.397,Z 1109.546,A -85,B 0,C 180,E1 20730.493,E2 20730.493} C_VEL
LIN {X 0,Y 379.124,Z 1169.931,A -85,B 0,C 180,E1 20737.812,E2 20737.812} C_VEL
LIN {X 0,Y 348.065,Z 1219.487,A -85,B 0,C 180,E1 20747.941,E2 20747.941} C_VEL
LIN {X 0,Y 326.258,Z 1255.915,A -85,B 0,C 180,E1 20760.786,E2 20760.786} C_VEL
LIN {X 0,Y 316.623,Z 1277.477,A -85,B 0,C 180,E1 20774.726,E2 20774.726} C_VEL
LIN {X 0,Y 315.14,Z 1284.82,A -85,B 0,C 180,E1 20785.86,E2 20785.86} C_VEL
LIN {X 0,Y 315.144,Z 1283.776,A -85,B 0,C 180,E1 20796.91,E2 20796.91} C_VEL
LIN {X 0,Y 318.408,Z 1272.477,A -85,B 0,C 180,E1 20809.475,E2 20809.475} C_VEL
LIN {X 0,Y 330.397,Z 1248.185,A -85,B 0,C 180,E1 20822.638,E2 20822.638} C_VEL
LIN {X 0,Y 354.987,Z 1208.576,A -85,B 0,C 180,E1 20834.821,E2 20834.821} C_VEL
LIN {X 0,Y 387.592,Z 1155.54,A -85,B 0,C 180,E1 20844.329,E2 20844.329} C_VEL
LIN {X 0,Y 420.483,Z 1093.118,A -85,B 0,C 180,E1 20850.939,E2 20850.939} C_VEL
LIN {X 0,Y 442.753,Z 1038.568,A -85,B 0,C 180,E1 20854.676,E2 20854.676} C_VEL
LIN {X 0,Y 434.206,Z 1006.765,A -85,B 0,C 180,E1 20862.758,E2 20862.758} C_VEL
LIN {X 0,Y 433.808,Z 1005.675,A -85,B 0,C 180,E1 20863.12,E2 20863.12} C_VEL
LIN {X 0,Y 426.517,Z 1001.064,A -85,B 0,C 180,E1 20867.731,E2 20867.731} C_VEL
LIN {X 0,Y 422.56,Z 990.001,A -85,B 0,C 180,E1 20874.884,E2 20874.884} C_VEL
LIN {X 0,Y 421.852,Z 987.231,A -85,B 0,C 180,E1 20881.064,E2 20881.064} C_VEL
LIN {X 0,Y 424.71,Z 997.029,A -85,B 0,C 180,E1 20890.426,E2 20890.426} C_VEL
LIN {X 0,Y 431.414,Z 1019.496,A -85,B 0,C 180,E1 20899.016,E2 20899.016} C_VEL
LIN {X 0,Y 436.053,Z 1045.39,A -85,B 0,C 180,E1 20905.183,E2 20905.183} C_VEL
LIN {X 0,Y 405.315,Z 1112.02,A -85,B 0,C 180,E1 20910.252,E2 20910.252} C_VEL
LIN {X 0,Y 370.91,Z 1170.945,A -85,B 0,C 180,E1 20917.858,E2 20917.858} C_VEL
LIN {X 0,Y 339.519,Z 1218.624,A -85,B 0,C 180,E1 20928.427,E2 20928.427} C_VEL
LIN {X 0,Y 317.936,Z 1252.366,A -85,B 0,C 180,E1 20941.408,E2 20941.408} C_VEL
LIN {X 0,Y 308.78,Z 1270.944,A -85,B 0,C 180,E1 20954.328,E2 20954.328} C_VEL
LIN {X 0,Y 307.068,Z 1278.051,A -85,B 0,C 180,E1 20965.752,E2 20965.752} C_VEL
LIN {X 0,Y 307.306,Z 1276.996,A -85,B 0,C 180,E1 20977.087,E2 20977.087} C_VEL
LIN {X 0,Y 310.713,Z 1265.924,A -85,B 0,C 180,E1 20989.978,E2 20989.978} C_VEL
LIN {X 0,Y 325.131,Z 1240.326,A -85,B 0,C 180,E1 21004.037,E2 21004.037} C_VEL
LIN {X 0,Y 351.398,Z 1200.711,A -85,B 0,C 180,E1 21016.155,E2 21016.155} C_VEL
LIN {X 0,Y 384.55,Z 1148.665,A -85,B 0,C 180,E1 21025.409,E2 21025.409} C_VEL
LIN {X 0,Y 418.091,Z 1086.364,A -85,B 0,C 180,E1 21031.915,E2 21031.915} C_VEL
LIN {X 0,Y 436.33,Z 1043.196,A -85,B 0,C 180,E1 21034.985,E2 21034.985} C_VEL
LIN {X 0,Y 429.443,Z 1012.323,A -85,B 0,C 180,E1 21043.022,E2 21043.022} C_VEL
LIN {X 0,Y 423.57,Z 992.56,A -85,B 0,C 180,E1 21051.73,E2 21051.73} C_VEL
LIN {X 0,Y 422.011,Z 986.032,A -85,B 0,C 180,E1 21058.937,E2 21058.937} C_VEL
LIN {X 0,Y 424.333,Z 994.921,A -85,B 0,C 180,E1 21069.224,E2 21069.224} C_VEL
LIN {X 0,Y 431.16,Z 1016.34,A -85,B 0,C 180,E1 21077.896,E2 21077.896} C_VEL
LIN {X 0,Y 437.555,Z 1043.692,A -85,B 0,C 180,E1 21084.714,E2 21084.714} C_VEL
LIN {X 0,Y 406.052,Z 1113.75,A -85,B 0,C 180,E1 21089.886,E2 21089.886} C_VEL
LIN {X 0,Y 371.966,Z 1173.224,A -85,B 0,C 180,E1 21097.342,E2 21097.342} C_VEL
LIN {X 0,Y 340.475,Z 1221.446,A -85,B 0,C 180,E1 21107.566,E2 21107.566} C_VEL
LIN {X 0,Y 318.29,Z 1257.006,A -85,B 0,C 180,E1 21120.66,E2 21120.66} C_VEL
LIN {X 0,Y 308.761,Z 1277.387,A -85,B 0,C 180,E1 21134.327,E2 21134.327} C_VEL
LIN {X 0,Y 307.135,Z 1284.732,A -85,B 0,C 180,E1 21145.752,E2 21145.752} C_VEL
LIN {X 0,Y 307.141,Z 1283.688,A -85,B 0,C 180,E1 21157.091,E2 21157.091} C_VEL
LIN {X 0,Y 310.632,Z 1272.388,A -85,B 0,C 180,E1 21169.983,E2 21169.983} C_VEL
LIN {X 0,Y 323.355,Z 1248.094,A -85,B 0,C 180,E1 21183.441,E2 21183.441} C_VEL
LIN {X 0,Y 349.063,Z 1208.486,A -85,B 0,C 180,E1 21195.795,E2 21195.795} C_VEL
LIN {X 0,Y 382.693,Z 1155.645,A -85,B 0,C 180,E1 21205.314,E2 21205.314} C_VEL
LIN {X 0,Y 416.087,Z 1094.04,A -85,B 0,C 180,E1 21211.848,E2 21211.848} C_VEL
LIN {X 0,Y 437.753,Z 1042.313,A -85,B 0,C 180,E1 21215.489,E2 21215.489} C_VEL
LIN {X 0,Y 429.895,Z 1011.705,A -85,B 0,C 180,E1 21223.636,E2 21223.636} C_VEL
LIN {X 0,Y 426.517,Z 1001.064,A -85,B 0,C 180,E1 21227.731,E2 21227.731} C_VEL
LIN {X 0,Y 420.606,Z 1000.146,A -85,B 0,C 180,E1 21232.487,E2 21232.487} C_VEL
LIN {X 0,Y 418.949,Z 994.688,A -85,B 0,C 180,E1 21241.071,E2 21241.071} C_VEL
LIN {X 0,Y 421.11,Z 1002.76,A -85,B 0,C 180,E1 21249.363,E2 21249.363} C_VEL
LIN {X 0,Y 426.98,Z 1024.165,A -85,B 0,C 180,E1 21258.147,E2 21258.147} C_VEL
LIN {X 0,Y 431.019,Z 1049.435,A -85,B 0,C 180,E1 21264.439,E2 21264.439} C_VEL
LIN {X 0,Y 399.818,Z 1114.674,A -85,B 0,C 180,E1 21269.496,E2 21269.496} C_VEL
LIN {X 0,Y 364.587,Z 1172.951,A -85,B 0,C 180,E1 21277.158,E2 21277.158} C_VEL
LIN {X 0,Y 332.446,Z 1219.912,A -85,B 0,C 180,E1 21287.828,E2 21287.828} C_VEL
LIN {X 0,Y 310.564,Z 1252.631,A -85,B 0,C 180,E1 21300.77,E2 21300.77} C_VEL
LIN {X 0,Y 300.443,Z 1272.333,A -85,B 0,C 180,E1 21315.382,E2 21315.382} C_VEL
LIN {X 0,Y 299.062,Z 1278.139,A -85,B 0,C 180,E1 21325.638,E2 21325.638} C_VEL
LIN {X 0,Y 299.305,Z 1277.084,A -85,B 0,C 180,E1 21337.277,E2 21337.277} C_VEL
LIN {X 0,Y 303.038,Z 1266.014,A -85,B 0,C 180,E1 21350.506,E2 21350.506} C_VEL
LIN {X 0,Y 318.27,Z 1240.418,A -85,B 0,C 180,E1 21364.875,E2 21364.875} C_VEL
LIN {X 0,Y 346.371,Z 1199.825,A -85,B 0,C 180,E1 21377.37,E2 21377.37} C_VEL
LIN {X 0,Y 381.076,Z 1146.838,A -85,B 0,C 180,E1 21386.691,E2 21386.691} C_VEL
LIN {X 0,Y 415.551,Z 1083.877,A -85,B 0,C 180,E1 21393.111,E2 21393.111} C_VEL
LIN {X 0,Y 431.292,Z 1047.238,A -85,B 0,C 180,E1 21395.739,E2 21395.739} C_VEL
LIN {X 0,Y 425.252,Z 1017.208,A -85,B 0,C 180,E1 21403.916,E2 21403.916} C_VEL
LIN {X 0,Y 420.222,Z 998.669,A -85,B 0,C 180,E1 21412.707,E2 21412.707} C_VEL
LIN {X 0,Y 418.903,Z 994.214,A -85,B 0,C 180,E1 21421.004,E2 21421.004} C_VEL
LIN {X 0,Y 422.012,Z 1004.417,A -85,B 0,C 180,E1 21430.321,E2 21430.321} C_VEL
LIN {X 0,Y 428.729,Z 1028.362,A -85,B 0,C 180,E1 21439.207,E2 21439.207} C_VEL
LIN {X 0,Y 432.315,Z 1048.589,A -85,B 0,C 180,E1 21444.066,E2 21444.066} C_VEL
LIN {X 0,Y 399.844,Z 1117.481,A -85,B 0,C 180,E1 21449.232,E2 21449.232} C_VEL
LIN {X 0,Y 364.786,Z 1176.356,A -85,B 0,C 180,E1 21456.844,E2 21456.844} C_VEL
LIN {X 0,Y 332.733,Z 1223.583,A -85,B 0,C 180,E1 21467.247,E2 21467.247} C_VEL
LIN {X 0,Y 310.133,Z 1258.45,A -85,B 0,C 180,E1 21480.725,E2 21480.725} C_VEL
LIN {X 0,Y 300.391,Z 1278.646,A -85,B 0,C 180,E1 21495.379,E2 21495.379} C_VEL
LIN {X 0,Y 299.12,Z 1284.644,A -85,B 0,C 180,E1 21505.638,E2 21505.638} C_VEL
LIN {X 0,Y 299.14,Z 1283.6,A -85,B 0,C 180,E1 21517.281,E2 21517.281} C_VEL
LIN {X 0,Y 302.888,Z 1272.298,A -85,B 0,C 180,E1 21530.517,E2 21530.517} C_VEL
LIN {X 0,Y 316.399,Z 1248.004,A -85,B 0,C 180,E1 21544.277,E2 21544.277} C_VEL
LIN {X 0,Y 343.406,Z 1208.201,A -85,B 0,C 180,E1 21556.842,E2 21556.842} C_VEL
LIN {X 0,Y 378.025,Z 1155.557,A -85,B 0,C 180,E1 21566.35,E2 21566.35} C_VEL
LIN {X 0,Y 412.248,Z 1094.021,A -85,B 0,C 180,E1 21572.848,E2 21572.848} C_VEL
LIN {X 0,Y 432.734,Z 1046.353,A -85,B 0,C 180,E1 21576.26,E2 21576.26} C_VEL
LIN {X 0,Y 425.667,Z 1016.676,A -85,B 0,C 180,E1 21584.531,E2 21584.531} C_VEL
LIN {X 0,Y 420.606,Z 1000.146,A -85,B 0,C 180,E1 21592.487,E2 21592.487} C_VEL
LIN {X 0,Y 416.195,Z 1003.036,A -85,B 0,C 180,E1 21597.299,E2 21597.299} C_VEL
LIN {X 0,Y 416.563,Z 1004.814,A -85,B 0,C 180,E1 21605.258,E2 21605.258} C_VEL
LIN {X 0,Y 420.598,Z 1020.504,A -85,B 0,C 180,E1 21614.288,E2 21614.288} C_VEL
LIN {X 0,Y 425.842,Z 1047.628,A -85,B 0,C 180,E1 21622.476,E2 21622.476} C_VEL
LIN {X 0,Y 425.375,Z 1055.156,A -85,B 0,C 180,E1 21623.779,E2 21623.779} C_VEL
LIN {X 0,Y 392.54,Z 1120.63,A -85,B 0,C 180,E1 21629.05,E2 21629.05} C_VEL
LIN {X 0,Y 356.401,Z 1177.835,A -85,B 0,C 180,E1 21636.939,E2 21636.939} C_VEL
LIN {X 0,Y 324.115,Z 1223.097,A -85,B 0,C 180,E1 21647.791,E2 21647.791} C_VEL
LIN {X 0,Y 301.053,Z 1256.274,A -85,B 0,C 180,E1 21661.965,E2 21661.965} C_VEL
LIN {X 0,Y 292.167,Z 1273.617,A -85,B 0,C 180,E1 21676.492,E2 21676.492} C_VEL
LIN {X 0,Y 291.027,Z 1278.661,A -85,B 0,C 180,E1 21688.507,E2 21688.507} C_VEL
LIN {X 0,Y 291.662,Z 1275.582,A -85,B 0,C 180,E1 21700.486,E2 21700.486} C_VEL
LIN {X 0,Y 298.909,Z 1259.961,A -85,B 0,C 180,E1 21715.547,E2 21715.547} C_VEL
LIN {X 0,Y 319,Z 1229.688,A -85,B 0,C 180,E1 21729.926,E2 21729.926} C_VEL
LIN {X 0,Y 351.045,Z 1185.409,A -85,B 0,C 180,E1 21741.51,E2 21741.51} C_VEL
LIN {X 0,Y 386.923,Z 1129.893,A -85,B 0,C 180,E1 21749.853,E2 21749.853} C_VEL
LIN {X 0,Y 420.82,Z 1065.127,A -85,B 0,C 180,E1 21755.471,E2 21755.471} C_VEL
LIN {X 0,Y 426.208,Z 1050.432,A -85,B 0,C 180,E1 21756.712,E2 21756.712} C_VEL
LIN {X 0,Y 421.158,Z 1022.558,A -85,B 0,C 180,E1 21764.72,E2 21764.72} C_VEL
LIN {X 0,Y 417.213,Z 1006.253,A -85,B 0,C 180,E1 21772.654,E2 21772.654} C_VEL
LIN {X 0,Y 415.991,Z 1001.696,A -85,B 0,C 180,E1 21781.011,E2 21781.011} C_VEL
LIN {X 0,Y 418.765,Z 1012.084,A -85,B 0,C 180,E1 21790.401,E2 21790.401} C_VEL
LIN {X 0,Y 424.848,Z 1036.002,A -85,B 0,C 180,E1 21799.265,E2 21799.265} C_VEL
LIN {X 0,Y 426.669,Z 1054.214,A -85,B 0,C 180,E1 21803.403,E2 21803.403} C_VEL
LIN {X 0,Y 393.347,Z 1121.899,A -85,B 0,C 180,E1 21808.637,E2 21808.637} C_VEL
LIN {X 0,Y 357.661,Z 1179.483,A -85,B 0,C 180,E1 21816.33,E2 21816.33} C_VEL
LIN {X 0,Y 324.175,Z 1226.939,A -85,B 0,C 180,E1 21827.287,E2 21827.287} C_VEL
LIN {X 0,Y 301.363,Z 1261.063,A -85,B 0,C 180,E1 21841.441,E2 21841.441} C_VEL
LIN {X 0,Y 292.066,Z 1279.784,A -85,B 0,C 180,E1 21856.487,E2 21856.487} C_VEL
LIN {X 0,Y 291.005,Z 1285.019,A -85,B 0,C 180,E1 21868.507,E2 21868.507} C_VEL
LIN {X 0,Y 291.509,Z 1281.891,A -85,B 0,C 180,E1 21880.491,E2 21880.491} C_VEL
LIN {X 0,Y 297.443,Z 1267.613,A -85,B 0,C 180,E1 21894.524,E2 21894.524} C_VEL
LIN {X 0,Y 315.8,Z 1239.11,A -85,B 0,C 180,E1 21908.63,E2 21908.63} C_VEL
LIN {X 0,Y 346.807,Z 1195.393,A -85,B 0,C 180,E1 21920.687,E2 21920.687} C_VEL
LIN {X 0,Y 383.149,Z 1139.736,A -85,B 0,C 180,E1 21929.416,E2 21929.416} C_VEL
LIN {X 0,Y 417.38,Z 1075.766,A -85,B 0,C 180,E1 21935.216,E2 21935.216} C_VEL
LIN {X 0,Y 427.802,Z 1050.969,A -85,B 0,C 180,E1 21936.905,E2 21936.905} C_VEL
LIN {X 0,Y 421.884,Z 1023.162,A -85,B 0,C 180,E1 21944.923,E2 21944.923} C_VEL
LIN {X 0,Y 417.125,Z 1006.004,A -85,B 0,C 180,E1 21953.77,E2 21953.77} C_VEL
LIN {X 0,Y 416.195,Z 1003.036,A -85,B 0,C 180,E1 21957.299,E2 21957.299} C_VEL
LIN {X 0,Y 412.885,Z 1010.053,A -85,B 0,C 180,E1 21962.113,E2 21962.113} C_VEL
LIN {X 0,Y 415.338,Z 1020.756,A -85,B 0,C 180,E1 21971.09,E2 21971.09} C_VEL
LIN {X 0,Y 419.943,Z 1043.85,A -85,B 0,C 180,E1 21979.557,E2 21979.557} C_VEL
LIN {X 0,Y 421.017,Z 1057.95,A -85,B 0,C 180,E1 21982.93,E2 21982.93} C_VEL
LIN {X 0,Y 386.605,Z 1124.184,A -85,B 0,C 180,E1 21988.339,E2 21988.339} C_VEL
LIN {X 0,Y 348.966,Z 1181.419,A -85,B 0,C 180,E1 21996.489,E2 21996.489} C_VEL
LIN {X 0,Y 315.87,Z 1225.87,A -85,B 0,C 180,E1 22007.634,E2 22007.634} C_VEL
LIN {X 0,Y 293.55,Z 1256.745,A -85,B 0,C 180,E1 22021.427,E2 22021.427} C_VEL
LIN {X 0,Y 284.275,Z 1273.705,A -85,B 0,C 180,E1 22036.11,E2 22036.11} C_VEL
LIN {X 0,Y 283.021,Z 1278.748,A -85,B 0,C 180,E1 22048.465,E2 22048.465} C_VEL
LIN {X 0,Y 283.711,Z 1275.671,A -85,B 0,C 180,E1 22060.783,E2 22060.783} C_VEL
LIN {X 0,Y 291.409,Z 1260.053,A -85,B 0,C 180,E1 22076.254,E2 22076.254} C_VEL
LIN {X 0,Y 312.632,Z 1229.781,A -85,B 0,C 180,E1 22090.91,E2 22090.91} C_VEL
LIN {X 0,Y 346.246,Z 1185.007,A -85,B 0,C 180,E1 22102.696,E2 22102.696} C_VEL
LIN {X 0,Y 383.481,Z 1128.939,A -85,B 0,C 180,E1 22111.041,E2 22111.041} C_VEL
LIN {X 0,Y 418.164,Z 1063.743,A -85,B 0,C 180,E1 22116.594,E2 22116.594} C_VEL
LIN {X 0,Y 421.303,Z 1054.564,A -85,B 0,C 180,E1 22117.501,E2 22117.501} C_VEL
LIN {X 0,Y 416.8,Z 1027.315,A -85,B 0,C 180,E1 22125.743,E2 22125.743} C_VEL
LIN {X 0,Y 413.923,Z 1013.752,A -85,B 0,C 180,E1 22132.596,E2 22132.596} C_VEL
LIN {X 0,Y 412.916,Z 1009.091,A -85,B 0,C 180,E1 22141.018,E2 22141.018} C_VEL
LIN {X 0,Y 414.943,Z 1017.769,A -85,B 0,C 180,E1 22149.435,E2 22149.435} C_VEL
LIN {X 0,Y 420.218,Z 1040.547,A -85,B 0,C 180,E1 22158.393,E2 22158.393} C_VEL
LIN {X 0,Y 421.933,Z 1057.828,A -85,B 0,C 180,E1 22162.606,E2 22162.606} C_VEL
LIN {X 0,Y 387.335,Z 1125.527,A -85,B 0,C 180,E1 22167.941,E2 22167.941} C_VEL
LIN {X 0,Y 350.479,Z 1182.704,A -85,B 0,C 180,E1 22175.807,E2 22175.807} C_VEL
LIN {X 0,Y 316.569,Z 1228.912,A -85,B 0,C 180,E1 22186.896,E2 22186.896} C_VEL
LIN {X 0,Y 293.497,Z 1261.932,A -85,B 0,C 180,E1 22201.204,E2 22201.204} C_VEL
LIN {X 0,Y 284.162,Z 1279.694,A -85,B 0,C 180,E1 22216.104,E2 22216.104} C_VEL
LIN {X 0,Y 283.002,Z 1284.932,A -85,B 0,C 180,E1 22228.464,E2 22228.464} C_VEL
LIN {X 0,Y 283.543,Z 1281.802,A -85,B 0,C 180,E1 22240.789,E2 22240.789} C_VEL
LIN {X 0,Y 290.241,Z 1267.017,A -85,B 0,C 180,E1 22255.535,E2 22255.535} C_VEL
LIN {X 0,Y 310.723,Z 1237.054,A -85,B 0,C 180,E1 22270.292,E2 22270.292} C_VEL
LIN {X 0,Y 342.823,Z 1193.501,A -85,B 0,C 180,E1 22282.136,E2 22282.136} C_VEL
LIN {X 0,Y 380.263,Z 1137.536,A -85,B 0,C 180,E1 22290.739,E2 22290.739} C_VEL
LIN {X 0,Y 415.337,Z 1072.795,A -85,B 0,C 180,E1 22296.438,E2 22296.438} C_VEL
LIN {X 0,Y 422.883,Z 1055.319,A -85,B 0,C 180,E1 22297.631,E2 22297.631} C_VEL
LIN {X 0,Y 417.618,Z 1028.18,A -85,B 0,C 180,E1 22305.842,E2 22305.842} C_VEL
LIN {X 0,Y 413.518,Z 1012.408,A -85,B 0,C 180,E1 22314.772,E2 22314.772} C_VEL
LIN {X 0,Y 412.945,Z 1009.524,A -85,B 0,C 180,E1 22321.087,E2 22321.087} C_VEL
LIN {X 0,Y 412.885,Z 1010.053,A -85,B 0,C 180,E1 22322.113,E2 22322.113} C_VEL
LIN {X 0,Y 410.4,Z 1021.238,A -85,B 0,C 180,E1 22326.807,E2 22326.807} C_VEL
LIN {X 0,Y 413.808,Z 1038.913,A -85,B 0,C 180,E1 22335.627,E2 22335.627} C_VEL
LIN {X 0,Y 416.469,Z 1061.087,A -85,B 0,C 180,E1 22342.099,E2 22342.099} C_VEL
LIN {X 0,Y 381.661,Z 1125.992,A -85,B 0,C 180,E1 22347.441,E2 22347.441} C_VEL
LIN {X 0,Y 344.084,Z 1181.508,A -85,B 0,C 180,E1 22355.375,E2 22355.375} C_VEL
LIN {X 0,Y 309.543,Z 1226.234,A -85,B 0,C 180,E1 22366.694,E2 22366.694} C_VEL
LIN {X 0,Y 285.474,Z 1257.926,A -85,B 0,C 180,E1 22381.364,E2 22381.364} C_VEL
LIN {X 0,Y 276.364,Z 1273.794,A -85,B 0,C 180,E1 22395.704,E2 22395.704} C_VEL
LIN {X 0,Y 275.015,Z 1278.836,A -85,B 0,C 180,E1 22408.42,E2 22408.42} C_VEL
LIN {X 0,Y 275.756,Z 1275.76,A -85,B 0,C 180,E1 22421.098,E2 22421.098} C_VEL
LIN {X 0,Y 283.968,Z 1260.145,A -85,B 0,C 180,E1 22436.997,E2 22436.997} C_VEL
LIN {X 0,Y 306.359,Z 1229.874,A -85,B 0,C 180,E1 22451.934,E2 22451.934} C_VEL
LIN {X 0,Y 340.95,Z 1185.521,A -85,B 0,C 180,E1 22463.724,E2 22463.724} C_VEL
LIN {X 0,Y 378.9,Z 1130.081,A -85,B 0,C 180,E1 22472.012,E2 22472.012} C_VEL
LIN {X 0,Y 414.363,Z 1065.152,A -85,B 0,C 180,E1 22477.544,E2 22477.544} C_VEL
LIN {X 0,Y 416.37,Z 1057.524,A -85,B 0,C 180,E1 22478.595,E2 22478.595} C_VEL
LIN {X 0,Y 412.451,Z 1031.611,A -85,B 0,C 180,E1 22487.002,E2 22487.002} C_VEL
LIN {X 0,Y 409.891,Z 1019.271,A -85,B 0,C 180,E1 22494.656,E2 22494.656} C_VEL
LIN {X 0,Y 409.668,Z 1016.437,A -85,B 0,C 180,E1 22501.026,E2 22501.026} C_VEL
LIN {X 0,Y 411.607,Z 1025.327,A -85,B 0,C 180,E1 22509.512,E2 22509.512} C_VEL
LIN {X 0,Y 415.883,Z 1046.723,A -85,B 0,C 180,E1 22518.027,E2 22518.027} C_VEL
LIN {X 0,Y 416.706,Z 1062.658,A -85,B 0,C 180,E1 22521.87,E2 22521.87} C_VEL
LIN {X 0,Y 380.708,Z 1130.097,A -85,B 0,C 180,E1 22527.339,E2 22527.339} C_VEL
LIN {X 0,Y 342.407,Z 1187.1,A -85,B 0,C 180,E1 22535.527,E2 22535.527} C_VEL
LIN {X 0,Y 307.712,Z 1232.475,A -85,B 0,C 180,E1 22547.093,E2 22547.093} C_VEL
LIN {X 0,Y 284.448,Z 1264.43,A -85,B 0,C 180,E1 22562.084,E2 22562.084} C_VEL
LIN {X 0,Y 275.871,Z 1280.821,A -85,B 0,C 180,E1 22577.297,E2 22577.297} C_VEL
LIN {X 0,Y 275.01,Z 1284.844,A -85,B 0,C 180,E1 22588.42,E2 22588.42} C_VEL
LIN {X 0,Y 275.574,Z 1281.714,A -85,B 0,C 180,E1 22601.105,E2 22601.105} C_VEL
LIN {X 0,Y 282.803,Z 1266.927,A -85,B 0,C 180,E1 22616.257,E2 22616.257} C_VEL
LIN {X 0,Y 304.361,Z 1236.963,A -85,B 0,C 180,E1 22631.315,E2 22631.315} C_VEL
LIN {X 0,Y 338.025,Z 1193.078,A -85,B 0,C 180,E1 22643.317,E2 22643.317} C_VEL
LIN {X 0,Y 375.893,Z 1138.038,A -85,B 0,C 180,E1 22651.779,E2 22651.779} C_VEL
LIN {X 0,Y 411.298,Z 1074.493,A -85,B 0,C 180,E1 22657.364,E2 22657.364} C_VEL
LIN {X 0,Y 417.98,Z 1059.024,A -85,B 0,C 180,E1 22658.524,E2 22658.524} C_VEL
LIN {X 0,Y 413.373,Z 1033.355,A -85,B 0,C 180,E1 22666.721,E2 22666.721} C_VEL
LIN {X 0,Y 410.266,Z 1019.791,A -85,B 0,C 180,E1 22674.73,E2 22674.73} C_VEL
LIN {X 0,Y 409.707,Z 1016.847,A -85,B 0,C 180,E1 22681.095,E2 22681.095} C_VEL
LIN {X 0,Y 410.4,Z 1021.238,A -85,B 0,C 180,E1 22686.807,E2 22686.807} C_VEL
LIN {X 0,Y 408.142,Z 1035.91,A -85,B 0,C 180,E1 22691.348,E2 22691.348} C_VEL
LIN {X 0,Y 411.354,Z 1059.889,A -85,B 0,C 180,E1 22699.931,E2 22699.931} C_VEL
LIN {X 0,Y 410.14,Z 1068.031,A -85,B 0,C 180,E1 22701.487,E2 22701.487} C_VEL
LIN {X 0,Y 373.873,Z 1132.367,A -85,B 0,C 180,E1 22707.031,E2 22707.031} C_VEL
LIN {X 0,Y 334.771,Z 1187.407,A -85,B 0,C 180,E1 22715.372,E2 22715.372} C_VEL
LIN {X 0,Y 299.269,Z 1231.263,A -85,B 0,C 180,E1 22727.379,E2 22727.379} C_VEL
LIN {X 0,Y 276.404,Z 1260.387,A -85,B 0,C 180,E1 22742.202,E2 22742.202} C_VEL
LIN {X 0,Y 268.095,Z 1275.059,A -85,B 0,C 180,E1 22756.923,E2 22756.923} C_VEL
LIN {X 0,Y 267.009,Z 1278.923,A -85,B 0,C 180,E1 22768.373,E2 22768.373} C_VEL
LIN {X 0,Y 267.833,Z 1275.849,A -85,B 0,C 180,E1 22781.431,E2 22781.431} C_VEL
LIN {X 0,Y 276.554,Z 1260.238,A -85,B 0,C 180,E1 22797.782,E2 22797.782} C_VEL
LIN {X 0,Y 300.197,Z 1229.967,A -85,B 0,C 180,E1 22813,E2 22813} C_VEL
LIN {X 0,Y 336.072,Z 1185.611,A -85,B 0,C 180,E1 22824.875,E2 22824.875} C_VEL
LIN {X 0,Y 375.724,Z 1129.251,A -85,B 0,C 180,E1 22833.219,E2 22833.219} C_VEL
LIN {X 0,Y 411.585,Z 1063.629,A -85,B 0,C 180,E1 22838.886,E2 22838.886} C_VEL
LIN {X 0,Y 408.741,Z 1039.266,A -85,B 0,C 180,E1 22846.882,E2 22846.882} C_VEL
LIN {X 0,Y 406.493,Z 1026.597,A -85,B 0,C 180,E1 22854.612,E2 22854.612} C_VEL
LIN {X 0,Y 406.428,Z 1023.755,A -85,B 0,C 180,E1 22861.035,E2 22861.035} C_VEL
LIN {X 0,Y 408.114,Z 1033.533,A -85,B 0,C 180,E1 22870.025,E2 22870.025} C_VEL
LIN {X 0,Y 412.005,Z 1056.565,A -85,B 0,C 180,E1 22878.799,E2 22878.799} C_VEL
LIN {X 0,Y 411.424,Z 1067.379,A -85,B 0,C 180,E1 22881.131,E2 22881.131} C_VEL
LIN {X 0,Y 374.79,Z 1133.383,A -85,B 0,C 180,E1 22886.589,E2 22886.589} C_VEL
LIN {X 0,Y 335.33,Z 1189.944,A -85,B 0,C 180,E1 22894.944,E2 22894.944} C_VEL
LIN {X 0,Y 299.606,Z 1234.851,A -85,B 0,C 180,E1 22906.895,E2 22906.895} C_VEL
LIN {X 0,Y 276.209,Z 1265.645,A -85,B 0,C 180,E1 22922.18,E2 22922.18} C_VEL
LIN {X 0,Y 267.959,Z 1280.732,A -85,B 0,C 180,E1 22936.916,E2 22936.916} C_VEL
LIN {X 0,Y 267.005,Z 1284.756,A -85,B 0,C 180,E1 22948.372,E2 22948.372} C_VEL
LIN {X 0,Y 267.618,Z 1281.625,A -85,B 0,C 180,E1 22961.44,E2 22961.44} C_VEL
LIN {X 0,Y 275.415,Z 1266.838,A -85,B 0,C 180,E1 22977.018,E2 22977.018} C_VEL
LIN {X 0,Y 298.699,Z 1236.146,A -85,B 0,C 180,E1 22992.642,E2 22992.642} C_VEL
LIN {X 0,Y 333.101,Z 1192.989,A -85,B 0,C 180,E1 23004.47,E2 23004.47} C_VEL
LIN {X 0,Y 372.721,Z 1136.906,A -85,B 0,C 180,E1 23013.018,E2 23013.018} C_VEL
LIN {X 0,Y 409.405,Z 1071.948,A -85,B 0,C 180,E1 23018.58,E2 23018.58} C_VEL
LIN {X 0,Y 413.034,Z 1062.83,A -85,B 0,C 180,E1 23019.436,E2 23019.436} C_VEL
LIN {X 0,Y 408.926,Z 1037.146,A -85,B 0,C 180,E1 23028.262,E2 23028.262} C_VEL
LIN {X 0,Y 406.523,Z 1025.426,A -85,B 0,C 180,E1 23036.826,E2 23036.826} C_VEL
LIN {X 0,Y 406.381,Z 1025.304,A -85,B 0,C 180,E1 23043.245,E2 23043.245} C_VEL
LIN {X 0,Y 408.142,Z 1035.91,A -85,B 0,C 180,E1 23051.348,E2 23051.348} C_VEL
LIN {X 0,Y 405.563,Z 1053.665,A -85,B 0,C 180,E1 23055.694,E2 23055.694} C_VEL
LIN {X 0,Y 405.726,Z 1071.152,A -85,B 0,C 180,E1 23060.609,E2 23060.609} C_VEL
LIN {X 0,Y 368.52,Z 1135.026,A -85,B 0,C 180,E1 23066.184,E2 23066.184} C_VEL
LIN {X 0,Y 327.71,Z 1190.401,A -85,B 0,C 180,E1 23074.774,E2 23074.774} C_VEL
LIN {X 0,Y 291.35,Z 1233.476,A -85,B 0,C 180,E1 23087.055,E2 23087.055} C_VEL
LIN {X 0,Y 268.288,Z 1261.614,A -85,B 0,C 180,E1 23102.203,E2 23102.203} C_VEL
LIN {X 0,Y 259.83,Z 1275.996,A -85,B 0,C 180,E1 23118.213,E2 23118.213} C_VEL
LIN {X 0,Y 259.348,Z 1278.995,A -85,B 0,C 180,E1 23131.676,E2 23131.676} C_VEL
LIN {X 0,Y 261.03,Z 1273.11,A -85,B 0,C 180,E1 23146.286,E2 23146.286} C_VEL
LIN {X 0,Y 273.547,Z 1254.423,A -85,B 0,C 180,E1 23162.591,E2 23162.591} C_VEL
LIN {X 0,Y 301.782,Z 1221.116,A -85,B 0,C 180,E1 23177.2,E2 23177.2} C_VEL
LIN {X 0,Y 340.837,Z 1173.471,A -85,B 0,C 180,E1 23188.316,E2 23188.316} C_VEL
LIN {X 0,Y 380.6,Z 1115.918,A -85,B 0,C 180,E1 23195.71,E2 23195.71} C_VEL
LIN {X 0,Y 406.737,Z 1068.4,A -85,B 0,C 180,E1 23199.531,E2 23199.531} C_VEL
LIN {X 0,Y 404.441,Z 1043.853,A -85,B 0,C 180,E1 23208.059,E2 23208.059} C_VEL
LIN {X 0,Y 402.916,Z 1033.817,A -85,B 0,C 180,E1 23214.564,E2 23214.564} C_VEL
LIN {X 0,Y 402.861,Z 1030.954,A -85,B 0,C 180,E1 23221.044,E2 23221.044} C_VEL
LIN {X 0,Y 404.456,Z 1041.001,A -85,B 0,C 180,E1 23230.117,E2 23230.117} C_VEL
LIN {X 0,Y 407.615,Z 1064.56,A -85,B 0,C 180,E1 23239.01,E2 23239.01} C_VEL
LIN {X 0,Y 406.811,Z 1070.855,A -85,B 0,C 180,E1 23240.292,E2 23240.292} C_VEL
LIN {X 0,Y 368.953,Z 1136.712,A -85,B 0,C 180,E1 23245.833,E2 23245.833} C_VEL
LIN {X 0,Y 328.254,Z 1192.875,A -85,B 0,C 180,E1 23254.362,E2 23254.362} C_VEL
LIN {X 0,Y 291.982,Z 1236.627,A -85,B 0,C 180,E1 23266.462,E2 23266.462} C_VEL
LIN {X 0,Y 268.06,Z 1266.715,A -85,B 0,C 180,E1 23282.177,E2 23282.177} C_VEL
LIN {X 0,Y 259.674,Z 1281.525,A -85,B 0,C 180,E1 23298.205,E2 23298.205} C_VEL
LIN {X 0,Y 258.957,Z 1284.671,A -85,B 0,C 180,E1 23311.678,E2 23311.678} C_VEL
LIN {X 0,Y 260.5,Z 1279.442,A -85,B 0,C 180,E1 23325.187,E2 23325.187} C_VEL
LIN {X 0,Y 272.397,Z 1260.734,A -85,B 0,C 180,E1 23341.931,E2 23341.931} C_VEL
LIN {X 0,Y 300.289,Z 1226.632,A -85,B 0,C 180,E1 23357.078,E2 23357.078} C_VEL
LIN {X 0,Y 338.946,Z 1179.23,A -85,B 0,C 180,E1 23368.223,E2 23368.223} C_VEL
LIN {X 0,Y 379.611,Z 1120.058,A -85,B 0,C 180,E1 23375.928,E2 23375.928} C_VEL
LIN {X 0,Y 408.149,Z 1067.749,A -85,B 0,C 180,E1 23380.047,E2 23380.047} C_VEL
LIN {X 0,Y 404.995,Z 1043.545,A -85,B 0,C 180,E1 23388.694,E2 23388.694} C_VEL
LIN {X 0,Y 402.944,Z 1032.63,A -85,B 0,C 180,E1 23396.798,E2 23396.798} C_VEL
LIN {X 0,Y 402.825,Z 1032.993,A -85,B 0,C 180,E1 23403.922,E2 23403.922} C_VEL
LIN {X 0,Y 404.79,Z 1046.785,A -85,B 0,C 180,E1 23413.03,E2 23413.03} C_VEL
LIN {X 0,Y 405.563,Z 1053.665,A -85,B 0,C 180,E1 23415.694,E2 23415.694} C_VEL
LIN {X 0,Y 401.769,Z 1068.601,A -85,B 0,C 180,E1 23418.306,E2 23418.306} C_VEL
LIN {X 0,Y 400.475,Z 1076.169,A -85,B 0,C 180,E1 23419.851,E2 23419.851} C_VEL
LIN {X 0,Y 362.536,Z 1138.766,A -85,B 0,C 180,E1 23425.434,E2 23425.434} C_VEL
LIN {X 0,Y 320.677,Z 1193.345,A -85,B 0,C 180,E1 23434.147,E2 23434.147} C_VEL
LIN {X 0,Y 283.259,Z 1235.763,A -85,B 0,C 180,E1 23446.801,E2 23446.801} C_VEL
LIN {X 0,Y 260.158,Z 1262.84,A -85,B 0,C 180,E1 23462.203,E2 23462.203} C_VEL
LIN {X 0,Y 251.885,Z 1276.084,A -85,B 0,C 180,E1 23477.835,E2 23477.835} C_VEL
LIN {X 0,Y 251.333,Z 1279.083,A -85,B 0,C 180,E1 23491.729,E2 23491.729} C_VEL
LIN {X 0,Y 253.183,Z 1273.2,A -85,B 0,C 180,E1 23506.806,E2 23506.806} C_VEL
LIN {X 0,Y 265.667,Z 1255.658,A -85,B 0,C 180,E1 23522.84,E2 23522.84} C_VEL
LIN {X 0,Y 294.438,Z 1223.158,A -85,B 0,C 180,E1 23537.766,E2 23537.766} C_VEL
LIN {X 0,Y 334.048,Z 1176.752,A -85,B 0,C 180,E1 23548.971,E2 23548.971} C_VEL
LIN {X 0,Y 375.146,Z 1119.459,A -85,B 0,C 180,E1 23556.513,E2 23556.513} C_VEL
LIN {X 0,Y 401.851,Z 1071.984,A -85,B 0,C 180,E1 23560.545,E2 23560.545} C_VEL
LIN {X 0,Y 400.217,Z 1048.933,A -85,B 0,C 180,E1 23569.039,E2 23569.039} C_VEL
LIN {X 0,Y 399.095,Z 1039.166,A -85,B 0,C 180,E1 23576.985,E2 23576.985} C_VEL
LIN {X 0,Y 399.272,Z 1039.487,A -85,B 0,C 180,E1 23583.232,E2 23583.232} C_VEL
LIN {X 0,Y 401.024,Z 1051.895,A -85,B 0,C 180,E1 23591.973,E2 23591.973} C_VEL
LIN {X 0,Y 402.973,Z 1072.781,A -85,B 0,C 180,E1 23599.302,E2 23599.302} C_VEL
LIN {X 0,Y 364.192,Z 1138.472,A -85,B 0,C 180,E1 23604.869,E2 23604.869} C_VEL
LIN {X 0,Y 322.951,Z 1193.577,A -85,B 0,C 180,E1 23613.295,E2 23613.295} C_VEL
LIN {X 0,Y 285.709,Z 1236.787,A -85,B 0,C 180,E1 23625.392,E2 23625.392} C_VEL
LIN {X 0,Y 260.76,Z 1266.623,A -85,B 0,C 180,E1 23641.327,E2 23641.327} C_VEL
LIN {X 0,Y 251.729,Z 1281.436,A -85,B 0,C 180,E1 23657.827,E2 23657.827} C_VEL
LIN {X 0,Y 250.951,Z 1284.583,A -85,B 0,C 180,E1 23671.731,E2 23671.731} C_VEL
LIN {X 0,Y 252.662,Z 1279.354,A -85,B 0,C 180,E1 23685.67,E2 23685.67} C_VEL
LIN {X 0,Y 265.305,Z 1260.643,A -85,B 0,C 180,E1 23702.89,E2 23702.89} C_VEL
LIN {X 0,Y 294.633,Z 1226.542,A -85,B 0,C 180,E1 23718.274,E2 23718.274} C_VEL
LIN {X 0,Y 334.623,Z 1179.141,A -85,B 0,C 180,E1 23729.439,E2 23729.439} C_VEL
LIN {X 0,Y 375.878,Z 1120.695,A -85,B 0,C 180,E1 23737.003,E2 23737.003} C_VEL
LIN {X 0,Y 403.254,Z 1072.194,A -85,B 0,C 180,E1 23740.818,E2 23740.818} C_VEL
LIN {X 0,Y 400.672,Z 1048.783,A -85,B 0,C 180,E1 23749.675,E2 23749.675} C_VEL
LIN {X 0,Y 399.529,Z 1038.21,A -85,B 0,C 180,E1 23758.947,E2 23758.947} C_VEL
LIN {X 0,Y 399.618,Z 1044.157,A -85,B 0,C 180,E1 23767.671,E2 23767.671} C_VEL
LIN {X 0,Y 401.343,Z 1061.338,A -85,B 0,C 180,E1 23775.886,E2 23775.886} C_VEL
LIN {X 0,Y 401.769,Z 1068.601,A -85,B 0,C 180,E1 23778.306,E2 23778.306} C_VEL
LIN {X 0,Y 397.873,Z 1077.46,A -85,B 0,C 180,E1 23779.157,E2 23779.157} C_VEL
LIN {X 0,Y 391.074,Z 1088.245,A -85,B 0,C 180,E1 23779.564,E2 23779.564} C_VEL
LIN {X 0,Y 350.872,Z 1150.105,A -85,B 0,C 180,E1 23785.649,E2 23785.649} C_VEL
LIN {X 0,Y 308.814,Z 1201.564,A -85,B 0,C 180,E1 23794.755,E2 23794.755} C_VEL
LIN {X 0,Y 272.056,Z 1241.277,A -85,B 0,C 180,E1 23808.016,E2 23808.016} C_VEL
LIN {X 0,Y 250.234,Z 1266.228,A -85,B 0,C 180,E1 23824.351,E2 23824.351} C_VEL
LIN {X 0,Y 243.326,Z 1277.738,A -85,B 0,C 180,E1 23841.036,E2 23841.036} C_VEL
LIN {X 0,Y 243.151,Z 1278.718,A -85,B 0,C 180,E1 23855.368,E2 23855.368} C_VEL
LIN {X 0,Y 247.439,Z 1270.009,A -85,B 0,C 180,E1 23871.576,E2 23871.576} C_VEL
LIN {X 0,Y 266.444,Z 1247.383,A -85,B 0,C 180,E1 23888.763,E2 23888.763} C_VEL
LIN {X 0,Y 301.156,Z 1210.067,A -85,B 0,C 180,E1 23902.917,E2 23902.917} C_VEL
LIN {X 0,Y 343.032,Z 1160.213,A -85,B 0,C 180,E1 23912.862,E2 23912.862} C_VEL
LIN {X 0,Y 384.585,Z 1099.169,A -85,B 0,C 180,E1 23919.478,E2 23919.478} C_VEL
LIN {X 0,Y 397.052,Z 1076.542,A -85,B 0,C 180,E1 23921.3,E2 23921.3} C_VEL
LIN {X 0,Y 396.1,Z 1055.223,A -85,B 0,C 180,E1 23929.482,E2 23929.482} C_VEL
LIN {X 0,Y 395.722,Z 1044.815,A -85,B 0,C 180,E1 23938.866,E2 23938.866} C_VEL
LIN {X 0,Y 396.036,Z 1051.193,A -85,B 0,C 180,E1 23947.669,E2 23947.669} C_VEL
LIN {X 0,Y 397.696,Z 1069.375,A -85,B 0,C 180,E1 23956.019,E2 23956.019} C_VEL
LIN {X 0,Y 397.159,Z 1079.056,A -85,B 0,C 180,E1 23958.619,E2 23958.619} C_VEL
LIN {X 0,Y 357.51,Z 1143.188,A -85,B 0,C 180,E1 23964.214,E2 23964.214} C_VEL
LIN {X 0,Y 315.574,Z 1196.977,A -85,B 0,C 180,E1 23972.755,E2 23972.755} C_VEL
LIN {X 0,Y 278.378,Z 1238.284,A -85,B 0,C 180,E1 23984.787,E2 23984.787} C_VEL
LIN {X 0,Y 252.466,Z 1267.881,A -85,B 0,C 180,E1 24001.439,E2 24001.439} C_VEL
LIN {X 0,Y 243.794,Z 1281.347,A -85,B 0,C 180,E1 24017.425,E2 24017.425} C_VEL
LIN {X 0,Y 242.948,Z 1284.495,A -85,B 0,C 180,E1 24031.788,E2 24031.788} C_VEL
LIN {X 0,Y 244.919,Z 1279.085,A -85,B 0,C 180,E1 24046.45,E2 24046.45} C_VEL
LIN {X 0,Y 258.293,Z 1260.552,A -85,B 0,C 180,E1 24063.902,E2 24063.902} C_VEL
LIN {X 0,Y 289.098,Z 1226.451,A -85,B 0,C 180,E1 24079.52,E2 24079.52} C_VEL
LIN {X 0,Y 330.137,Z 1179.422,A -85,B 0,C 180,E1 24090.63,E2 24090.63} C_VEL
LIN {X 0,Y 372.24,Z 1121.38,A -85,B 0,C 180,E1 24098.098,E2 24098.098} C_VEL
LIN {X 0,Y 398.419,Z 1076.231,A -85,B 0,C 180,E1 24101.728,E2 24101.728} C_VEL
LIN {X 0,Y 396.541,Z 1055.085,A -85,B 0,C 180,E1 24110.123,E2 24110.123} C_VEL
LIN {X 0,Y 395.808,Z 1045.32,A -85,B 0,C 180,E1 24118.938,E2 24118.938} C_VEL
LIN {X 0,Y 395.658,Z 1051.353,A -85,B 0,C 180,E1 24127.748,E2 24127.748} C_VEL
LIN {X 0,Y 396.885,Z 1069.167,A -85,B 0,C 180,E1 24136.168,E2 24136.168} C_VEL
LIN {X 0,Y 396.275,Z 1078.91,A -85,B 0,C 180,E1 24138.919,E2 24138.919} C_VEL
LIN {X 0,Y 391.074,Z 1088.245,A -85,B 0,C 180,E1 24139.564,E2 24139.564} C_VEL
LIN {X 0,Y 371.038,Z 1116.504,A -85,B 0,C 180,E1 24140.712,E2 24140.712} C_VEL
LIN {X 0,Y 328.224,Z 1174.233,A -85,B 0,C 180,E1 24147.972,E2 24147.972} C_VEL
LIN {X 0,Y 285.486,Z 1221.427,A -85,B 0,C 180,E1 24159.023,E2 24159.023} C_VEL
LIN {X 0,Y 253.787,Z 1254.087,A -85,B 0,C 180,E1 24173.895,E2 24173.895} C_VEL
LIN {X 0,Y 237.843,Z 1273.043,A -85,B 0,C 180,E1 24191.409,E2 24191.409} C_VEL
LIN {X 0,Y 235.067,Z 1278.84,A -85,B 0,C 180,E1 24204.447,E2 24204.447} C_VEL
LIN {X 0,Y 235.151,Z 1278.806,A -85,B 0,C 180,E1 24215.552,E2 24215.552} C_VEL
LIN {X 0,Y 239.761,Z 1270.174,A -85,B 0,C 180,E1 24232.21,E2 24232.21} C_VEL
LIN {X 0,Y 259.946,Z 1247.529,A -85,B 0,C 180,E1 24249.884,E2 24249.884} C_VEL
LIN {X 0,Y 296.502,Z 1209.85,A -85,B 0,C 180,E1 24264.286,E2 24264.286} C_VEL
LIN {X 0,Y 339.296,Z 1160.365,A -85,B 0,C 180,E1 24274.095,E2 24274.095} C_VEL
LIN {X 0,Y 381.792,Z 1099.263,A -85,B 0,C 180,E1 24280.629,E2 24280.629} C_VEL
LIN {X 0,Y 392.162,Z 1080.73,A -85,B 0,C 180,E1 24282.157,E2 24282.157} C_VEL
LIN {X 0,Y 391.881,Z 1060.129,A -85,B 0,C 180,E1 24290.688,E2 24290.688} C_VEL
LIN {X 0,Y 391.815,Z 1051.85,A -85,B 0,C 180,E1 24298.855,E2 24298.855} C_VEL
LIN {X 0,Y 392.073,Z 1058.391,A -85,B 0,C 180,E1 24307.747,E2 24307.747} C_VEL
LIN {X 0,Y 393.213,Z 1076.942,A -85,B 0,C 180,E1 24316.205,E2 24316.205} C_VEL
LIN {X 0,Y 392.184,Z 1083.277,A -85,B 0,C 180,E1 24317.783,E2 24317.783} C_VEL
LIN {X 0,Y 351.288,Z 1146.958,A -85,B 0,C 180,E1 24323.456,E2 24323.456} C_VEL
LIN {X 0,Y 308.045,Z 1200.212,A -85,B 0,C 180,E1 24332.198,E2 24332.198} C_VEL
LIN {X 0,Y 268.82,Z 1241.965,A -85,B 0,C 180,E1 24345.156,E2 24345.156} C_VEL
LIN {X 0,Y 243.567,Z 1269.598,A -85,B 0,C 180,E1 24362.162,E2 24362.162} C_VEL
LIN {X 0,Y 235.878,Z 1281.257,A -85,B 0,C 180,E1 24376.995,E2 24376.995} C_VEL
LIN {X 0,Y 234.952,Z 1284.408,A -85,B 0,C 180,E1 24391.849,E2 24391.849} C_VEL
LIN {X 0,Y 237.009,Z 1279.176,A -85,B 0,C 180,E1 24406.734,E2 24406.734} C_VEL
LIN {X 0,Y 251.377,Z 1260.462,A -85,B 0,C 180,E1 24424.968,E2 24424.968} C_VEL
LIN {X 0,Y 283.738,Z 1226.362,A -85,B 0,C 180,E1 24440.805,E2 24440.805} C_VEL
LIN {X 0,Y 325.665,Z 1179.889,A -85,B 0,C 180,E1 24451.816,E2 24451.816} C_VEL
LIN {X 0,Y 368.746,Z 1122.063,A -85,B 0,C 180,E1 24459.213,E2 24459.213} C_VEL
LIN {X 0,Y 393.546,Z 1080.969,A -85,B 0,C 180,E1 24462.441,E2 24462.441} C_VEL
LIN {X 0,Y 392.319,Z 1060.448,A -85,B 0,C 180,E1 24471.137,E2 24471.137} C_VEL
LIN {X 0,Y 391.905,Z 1052.351,A -85,B 0,C 180,E1 24478.927,E2 24478.927} C_VEL
LIN {X 0,Y 391.691,Z 1058.563,A -85,B 0,C 180,E1 24487.827,E2 24487.827} C_VEL
LIN {X 0,Y 392.309,Z 1076.692,A -85,B 0,C 180,E1 24496.319,E2 24496.319} C_VEL
LIN {X 0,Y 390.94,Z 1083.855,A -85,B 0,C 180,E1 24498.121,E2 24498.121} C_VEL
LIN {X 0,Y 371.038,Z 1116.504,A -85,B 0,C 180,E1 24500.712,E2 24500.712} C_VEL
LIN {X 0,Y 349.548,Z 1143.032,A -85,B 0,C 180,E1 24502.268,E2 24502.268} C_VEL
LIN {X 0,Y 305.075,Z 1195.971,A -85,B 0,C 180,E1 24510.815,E2 24510.815} C_VEL
LIN {X 0,Y 265.56,Z 1236.074,A -85,B 0,C 180,E1 24523.131,E2 24523.131} C_VEL
LIN {X 0,Y 237.62,Z 1263.972,A -85,B 0,C 180,E1 24540.222,E2 24540.222} C_VEL
LIN {X 0,Y 228.11,Z 1276.35,A -85,B 0,C 180,E1 24556.545,E2 24556.545} C_VEL
LIN {X 0,Y 227.32,Z 1279.346,A -85,B 0,C 180,E1 24571.912,E2 24571.912} C_VEL
LIN {X 0,Y 230.106,Z 1273.058,A -85,B 0,C 180,E1 24589.24,E2 24589.24} C_VEL
LIN {X 0,Y 246.739,Z 1254.242,A -85,B 0,C 180,E1 24607.122,E2 24607.122} C_VEL
LIN {X 0,Y 281.459,Z 1220.229,A -85,B 0,C 180,E1 24622.614,E2 24622.614} C_VEL
LIN {X 0,Y 324.767,Z 1173.636,A -85,B 0,C 180,E1 24633.359,E2 24633.359} C_VEL
LIN {X 0,Y 369.156,Z 1114.996,A -85,B 0,C 180,E1 24640.499,E2 24640.499} C_VEL
LIN {X 0,Y 387.321,Z 1085.417,A -85,B 0,C 180,E1 24642.879,E2 24642.879} C_VEL
LIN {X 0,Y 387.565,Z 1065.985,A -85,B 0,C 180,E1 24651.337,E2 24651.337} C_VEL
LIN {X 0,Y 387.899,Z 1058.901,A -85,B 0,C 180,E1 24658.843,E2 24658.843} C_VEL
LIN {X 0,Y 387.864,Z 1065.483,A -85,B 0,C 180,E1 24667.831,E2 24667.831} C_VEL
LIN {X 0,Y 388.412,Z 1084.6,A -85,B 0,C 180,E1 24676.472,E2 24676.472} C_VEL
LIN {X 0,Y 346.6,Z 1148.79,A -85,B 0,C 180,E1 24682.434,E2 24682.434} C_VEL
LIN {X 0,Y 301.862,Z 1202.029,A -85,B 0,C 180,E1 24691.288,E2 24691.288} C_VEL
LIN {X 0,Y 261.149,Z 1243.625,A -85,B 0,C 180,E1 24704.653,E2 24704.653} C_VEL
LIN {X 0,Y 236.278,Z 1269.506,A -85,B 0,C 180,E1 24721.224,E2 24721.224} C_VEL
LIN {X 0,Y 227.965,Z 1281.168,A -85,B 0,C 180,E1 24736.536,E2 24736.536} C_VEL
LIN {X 0,Y 226.944,Z 1284.32,A -85,B 0,C 180,E1 24751.915,E2 24751.915} C_VEL
LIN {X 0,Y 229.18,Z 1279.087,A -85,B 0,C 180,E1 24767.324,E2 24767.324} C_VEL
LIN {X 0,Y 244.541,Z 1260.371,A -85,B 0,C 180,E1 24786.096,E2 24786.096} C_VEL
LIN {X 0,Y 277.108,Z 1227.722,A -85,B 0,C 180,E1 24801.672,E2 24801.672} C_VEL
LIN {X 0,Y 320.871,Z 1180.908,A -85,B 0,C 180,E1 24812.941,E2 24812.941} C_VEL
LIN {X 0,Y 365.414,Z 1122.716,A -85,B 0,C 180,E1 24820.352,E2 24820.352} C_VEL
LIN {X 0,Y 388.638,Z 1084.656,A -85,B 0,C 180,E1 24823.504,E2 24823.504} C_VEL
LIN {X 0,Y 387.94,Z 1065.761,A -85,B 0,C 180,E1 24832.17,E2 24832.17} C_VEL
LIN {X 0,Y 387.996,Z 1059.393,A -85,B 0,C 180,E1 24838.916,E2 24838.916} C_VEL
LIN {X 0,Y 387.455,Z 1065.573,A -85,B 0,C 180,E1 24847.913,E2 24847.913} C_VEL
LIN {X 0,Y 387.426,Z 1083.977,A -85,B 0,C 180,E1 24856.459,E2 24856.459} C_VEL
LIN {X 0,Y 385.409,Z 1089.291,A -85,B 0,C 180,E1 24857.337,E2 24857.337} C_VEL
LIN {X 0,Y 349.548,Z 1143.032,A -85,B 0,C 180,E1 24862.268,E2 24862.268} C_VEL
LIN {X 0,Y 326.75,Z 1167.628,A -85,B 0,C 180,E1 24864.255,E2 24864.255} C_VEL
LIN {X 0,Y 280.675,Z 1216.407,A -85,B 0,C 180,E1 24874.638,E2 24874.638} C_VEL
LIN {X 0,Y 242.601,Z 1252.208,A -85,B 0,C 180,E1 24890.154,E2 24890.154} C_VEL
LIN {X 0,Y 223.487,Z 1271.92,A -85,B 0,C 180,E1 24908.086,E2 24908.086} C_VEL
LIN {X 0,Y 219.08,Z 1279.015,A -85,B 0,C 180,E1 24924.04,E2 24924.04} C_VEL
LIN {X 0,Y 219.153,Z 1278.983,A -85,B 0,C 180,E1 24935.958,E2 24935.958} C_VEL
LIN {X 0,Y 224.993,Z 1269.949,A -85,B 0,C 180,E1 24954.309,E2 24954.309} C_VEL
LIN {X 0,Y 248.621,Z 1246.578,A -85,B 0,C 180,E1 24972.987,E2 24972.987} C_VEL
LIN {X 0,Y 288.318,Z 1208.835,A -85,B 0,C 180,E1 24987.309,E2 24987.309} C_VEL
LIN {X 0,Y 333.843,Z 1158.806,A -85,B 0,C 180,E1 24996.91,E2 24996.91} C_VEL
LIN {X 0,Y 377.816,Z 1097.668,A -85,B 0,C 180,E1 25003.109,E2 25003.109} C_VEL
LIN {X 0,Y 382.596,Z 1089.227,A -85,B 0,C 180,E1 25003.92,E2 25003.92} C_VEL
LIN {X 0,Y 383.28,Z 1071.874,A -85,B 0,C 180,E1 25012,E2 25012} C_VEL
LIN {X 0,Y 383.709,Z 1065.783,A -85,B 0,C 180,E1 25018.831,E2 25018.831} C_VEL
LIN {X 0,Y 383.557,Z 1072.538,A -85,B 0,C 180,E1 25027.92,E2 25027.92} C_VEL
LIN {X 0,Y 383.527,Z 1089.569,A -85,B 0,C 180,E1 25035.796,E2 25035.796} C_VEL
LIN {X 0,Y 340.54,Z 1152.556,A -85,B 0,C 180,E1 25041.622,E2 25041.622} C_VEL
LIN {X 0,Y 294.95,Z 1204.713,A -85,B 0,C 180,E1 25050.545,E2 25050.545} C_VEL
LIN {X 0,Y 254.883,Z 1243.951,A -85,B 0,C 180,E1 25063.505,E2 25063.505} C_VEL
LIN {X 0,Y 229.077,Z 1269.415,A -85,B 0,C 180,E1 25080.23,E2 25080.23} C_VEL
LIN {X 0,Y 220.058,Z 1281.079,A -85,B 0,C 180,E1 25096.042,E2 25096.042} C_VEL
LIN {X 0,Y 219.019,Z 1284.231,A -85,B 0,C 180,E1 25108.016,E2 25108.016} C_VEL
LIN {X 0,Y 220.065,Z 1281.094,A -85,B 0,C 180,E1 25123.957,E2 25123.957} C_VEL
LIN {X 0,Y 233.126,Z 1265.135,A -85,B 0,C 180,E1 25143.569,E2 25143.569} C_VEL
LIN {X 0,Y 264.871,Z 1234.361,A -85,B 0,C 180,E1 25160.619,E2 25160.619} C_VEL
LIN {X 0,Y 308.947,Z 1189.906,A -85,B 0,C 180,E1 25172.633,E2 25172.633} C_VEL
LIN {X 0,Y 354.89,Z 1133.669,A -85,B 0,C 180,E1 25180.525,E2 25180.525} C_VEL
LIN {X 0,Y 383.772,Z 1088.789,A -85,B 0,C 180,E1 25184.478,E2 25184.478} C_VEL
LIN {X 0,Y 383.609,Z 1071.193,A -85,B 0,C 180,E1 25193.223,E2 25193.223} C_VEL
LIN {X 0,Y 383.59,Z 1066.455,A -85,B 0,C 180,E1 25201.17,E2 25201.17} C_VEL
LIN {X 0,Y 383.198,Z 1076.346,A -85,B 0,C 180,E1 25210.299,E2 25210.299} C_VEL
LIN {X 0,Y 382.2,Z 1090.844,A -85,B 0,C 180,E1 25216.268,E2 25216.268} C_VEL
LIN {X 0,Y 339.591,Z 1152,A -85,B 0,C 180,E1 25222.082,E2 25222.082} C_VEL
LIN {X 0,Y 326.75,Z 1167.628,A -85,B 0,C 180,E1 25224.255,E2 25224.255} C_VEL
LIN {X 0,Y 302.872,Z 1189.998,A -85,B 0,C 180,E1 25226.773,E2 25226.773} C_VEL
LIN {X 0,Y 258.267,Z 1232.765,A -85,B 0,C 180,E1 25238.919,E2 25238.919} C_VEL
LIN {X 0,Y 225.656,Z 1262.052,A -85,B 0,C 180,E1 25256.227,E2 25256.227} C_VEL
LIN {X 0,Y 212.316,Z 1276.527,A -85,B 0,C 180,E1 25275.523,E2 25275.523} C_VEL
LIN {X 0,Y 211.295,Z 1279.522,A -85,B 0,C 180,E1 25292.057,E2 25292.057} C_VEL
LIN {X 0,Y 214.696,Z 1273.238,A -85,B 0,C 180,E1 25310.682,E2 25310.682} C_VEL
LIN {X 0,Y 234.769,Z 1253.468,A -85,B 0,C 180,E1 25330.239,E2 25330.239} C_VEL
LIN {X 0,Y 272.608,Z 1219.477,A -85,B 0,C 180,E1 25345.733,E2 25345.733} C_VEL
LIN {X 0,Y 319.042,Z 1172.332,A -85,B 0,C 180,E1 25356.267,E2 25356.267} C_VEL
LIN {X 0,Y 364.802,Z 1114.038,A -85,B 0,C 180,E1 25363.033,E2 25363.033} C_VEL
LIN {X 0,Y 377.822,Z 1093.595,A -85,B 0,C 180,E1 25364.833,E2 25364.833} C_VEL
LIN {X 0,Y 378.982,Z 1077.311,A -85,B 0,C 180,E1 25373.065,E2 25373.065} C_VEL
LIN {X 0,Y 379.379,Z 1072.969,A -85,B 0,C 180,E1 25381.108,E2 25381.108} C_VEL
LIN {X 0,Y 379.116,Z 1082.365,A -85,B 0,C 180,E1 25389.757,E2 25389.757} C_VEL
LIN {X 0,Y 377.767,Z 1095.858,A -85,B 0,C 180,E1 25395.137,E2 25395.137} C_VEL
LIN {X 0,Y 333.035,Z 1158.125,A -85,B 0,C 180,E1 25401.012,E2 25401.012} C_VEL
LIN {X 0,Y 286.304,Z 1209.087,A -85,B 0,C 180,E1 25410.167,E2 25410.167} C_VEL
LIN {X 0,Y 244.084,Z 1248.515,A -85,B 0,C 180,E1 25424.396,E2 25424.396} C_VEL
LIN {X 0,Y 218.25,Z 1273.125,A -85,B 0,C 180,E1 25443.15,E2 25443.15} C_VEL
LIN {X 0,Y 211.337,Z 1282.621,A -85,B 0,C 180,E1 25459.665,E2 25459.665} C_VEL
LIN {X 0,Y 210.931,Z 1284.145,A -85,B 0,C 180,E1 25472.06,E2 25472.06} C_VEL
LIN {X 0,Y 213.583,Z 1278.909,A -85,B 0,C 180,E1 25488.634,E2 25488.634} C_VEL
LIN {X 0,Y 231.194,Z 1260.19,A -85,B 0,C 180,E1 25508.547,E2 25508.547} C_VEL
LIN {X 0,Y 267.358,Z 1227.145,A -85,B 0,C 180,E1 25524.651,E2 25524.651} C_VEL
LIN {X 0,Y 314.587,Z 1179.619,A -85,B 0,C 180,E1 25535.851,E2 25535.851} C_VEL
LIN {X 0,Y 360.531,Z 1122.087,A -85,B 0,C 180,E1 25542.856,E2 25542.856} C_VEL
LIN {X 0,Y 378.947,Z 1093.44,A -85,B 0,C 180,E1 25545.311,E2 25545.311} C_VEL
LIN {X 0,Y 379.301,Z 1078.178,A -85,B 0,C 180,E1 25553.146,E2 25553.146} C_VEL
LIN {X 0,Y 379.388,Z 1073.277,A -85,B 0,C 180,E1 25561.183,E2 25561.183} C_VEL
LIN {X 0,Y 378.588,Z 1082.292,A -85,B 0,C 180,E1 25569.843,E2 25569.843} C_VEL
LIN {X 0,Y 377.187,Z 1095.43,A -85,B 0,C 180,E1 25575.398,E2 25575.398} C_VEL
LIN {X 0,Y 333.56,Z 1155.762,A -85,B 0,C 180,E1 25581.246,E2 25581.246} C_VEL
LIN {X 0,Y 302.872,Z 1189.998,A -85,B 0,C 180,E1 25586.773,E2 25586.773} C_VEL
LIN {X 0,Y 278.422,Z 1210.143,A -85,B 0,C 180,E1 25589.937,E2 25589.937} C_VEL
LIN {X 0,Y 236.329,Z 1246.932,A -85,B 0,C 180,E1 25604.163,E2 25604.163} C_VEL
LIN {X 0,Y 210.031,Z 1270.256,A -85,B 0,C 180,E1 25623.885,E2 25623.885} C_VEL
LIN {X 0,Y 203.093,Z 1279.191,A -85,B 0,C 180,E1 25643.569,E2 25643.569} C_VEL
LIN {X 0,Y 203.16,Z 1279.159,A -85,B 0,C 180,E1 25656.429,E2 25656.429} C_VEL
LIN {X 0,Y 210.054,Z 1270.173,A -85,B 0,C 180,E1 25676.1,E2 25676.1} C_VEL
LIN {X 0,Y 236.934,Z 1246.491,A -85,B 0,C 180,E1 25695.918,E2 25695.918} C_VEL
LIN {X 0,Y 279.259,Z 1209.38,A -85,B 0,C 180,E1 25710.096,E2 25710.096} C_VEL
LIN {X 0,Y 327.215,Z 1159.55,A -85,B 0,C 180,E1 25719.501,E2 25719.501} C_VEL
LIN {X 0,Y 372.927,Z 1098.183,A -85,B 0,C 180,E1 25725.643,E2 25725.643} C_VEL
LIN {X 0,Y 374.475,Z 1082.813,A -85,B 0,C 180,E1 25734.149,E2 25734.149} C_VEL
LIN {X 0,Y 375.051,Z 1079.73,A -85,B 0,C 180,E1 25741.121,E2 25741.121} C_VEL
LIN {X 0,Y 374.434,Z 1089.347,A -85,B 0,C 180,E1 25749.881,E2 25749.881} C_VEL
LIN {X 0,Y 372.759,Z 1100.266,A -85,B 0,C 180,E1 25754.243,E2 25754.243} C_VEL
LIN {X 0,Y 327.088,Z 1161.564,A -85,B 0,C 180,E1 25760.137,E2 25760.137} C_VEL
LIN {X 0,Y 279.381,Z 1211.556,A -85,B 0,C 180,E1 25769.35,E2 25769.35} C_VEL
LIN {X 0,Y 235.826,Z 1250.481,A -85,B 0,C 180,E1 25784.096,E2 25784.096} C_VEL
LIN {X 0,Y 209.636,Z 1274.293,A -85,B 0,C 180,E1 25803.797,E2 25803.797} C_VEL
LIN {X 0,Y 203.027,Z 1283.586,A -85,B 0,C 180,E1 25823.567,E2 25823.567} C_VEL
LIN {X 0,Y 203.008,Z 1283.595,A -85,B 0,C 180,E1 25836.434,E2 25836.434} C_VEL
LIN {X 0,Y 208.701,Z 1275.343,A -85,B 0,C 180,E1 25854.847,E2 25854.847} C_VEL
LIN {X 0,Y 233.205,Z 1252.753,A -85,B 0,C 180,E1 25874.675,E2 25874.675} C_VEL
LIN {X 0,Y 275.508,Z 1215.295,A -85,B 0,C 180,E1 25889.687,E2 25889.687} C_VEL
LIN {X 0,Y 323.976,Z 1165.34,A -85,B 0,C 180,E1 25899.384,E2 25899.384} C_VEL
LIN {X 0,Y 369.275,Z 1105.923,A -85,B 0,C 180,E1 25905.368,E2 25905.368} C_VEL
LIN {X 0,Y 374.089,Z 1097.604,A -85,B 0,C 180,E1 25906.329,E2 25906.329} C_VEL
LIN {X 0,Y 374.784,Z 1083.543,A -85,B 0,C 180,E1 25914.23,E2 25914.23} C_VEL
LIN {X 0,Y 375.046,Z 1080.017,A -85,B 0,C 180,E1 25921.196,E2 25921.196} C_VEL
LIN {X 0,Y 373.918,Z 1089.258,A -85,B 0,C 180,E1 25929.967,E2 25929.967} C_VEL
LIN {X 0,Y 371.569,Z 1100.88,A -85,B 0,C 180,E1 25934.571,E2 25934.571} C_VEL
LIN {X 0,Y 326.503,Z 1160.602,A -85,B 0,C 180,E1 25940.546,E2 25940.546} C_VEL
LIN {X 0,Y 278.422,Z 1210.143,A -85,B 0,C 180,E1 25949.937,E2 25949.937} C_VEL
LIN {X 0,Y 254.088,Z 1227.944,A -85,B 0,C 180,E1 25953.968,E2 25953.968} C_VEL
LIN {X 0,Y 215.176,Z 1259.654,A -85,B 0,C 180,E1 25971.468,E2 25971.468} C_VEL
LIN {X 0,Y 197.348,Z 1275.857,A -85,B 0,C 180,E1 25992.099,E2 25992.099} C_VEL
LIN {X 0,Y 195.021,Z 1279.71,A -85,B 0,C 180,E1 26007.772,E2 26007.772} C_VEL
LIN {X 0,Y 196.692,Z 1276.652,A -85,B 0,C 180,E1 26025.656,E2 26025.656} C_VEL
LIN {X 0,Y 213.089,Z 1261.068,A -85,B 0,C 180,E1 26047.225,E2 26047.225} C_VEL
LIN {X 0,Y 250.38,Z 1230.808,A -85,B 0,C 180,E1 26064.854,E2 26064.854} C_VEL
LIN {X 0,Y 299.255,Z 1186.455,A -85,B 0,C 180,E1 26076.711,E2 26076.711} C_VEL
LIN {X 0,Y 347.978,Z 1131.018,A -85,B 0,C 180,E1 26084.053,E2 26084.053} C_VEL
LIN {X 0,Y 368.095,Z 1102.594,A -85,B 0,C 180,E1 26086.576,E2 26086.576} C_VEL
LIN {X 0,Y 369.898,Z 1089.574,A -85,B 0,C 180,E1 26094.077,E2 26094.077} C_VEL
LIN {X 0,Y 370.525,Z 1086.382,A -85,B 0,C 180,E1 26101.135,E2 26101.135} C_VEL
LIN {X 0,Y 369.66,Z 1096.297,A -85,B 0,C 180,E1 26110.006,E2 26110.006} C_VEL
LIN {X 0,Y 367.794,Z 1104.74,A -85,B 0,C 180,E1 26113.325,E2 26113.325} C_VEL
LIN {X 0,Y 321.204,Z 1164.995,A -85,B 0,C 180,E1 26119.219,E2 26119.219} C_VEL
LIN {X 0,Y 270.869,Z 1215.571,A -85,B 0,C 180,E1 26128.919,E2 26128.919} C_VEL
LIN {X 0,Y 226.944,Z 1252.98,A -85,B 0,C 180,E1 26144.083,E2 26144.083} C_VEL
